Yaskawa INFORM job: A_ROOF_SIDE_0617_2_PAINT_44.JBI

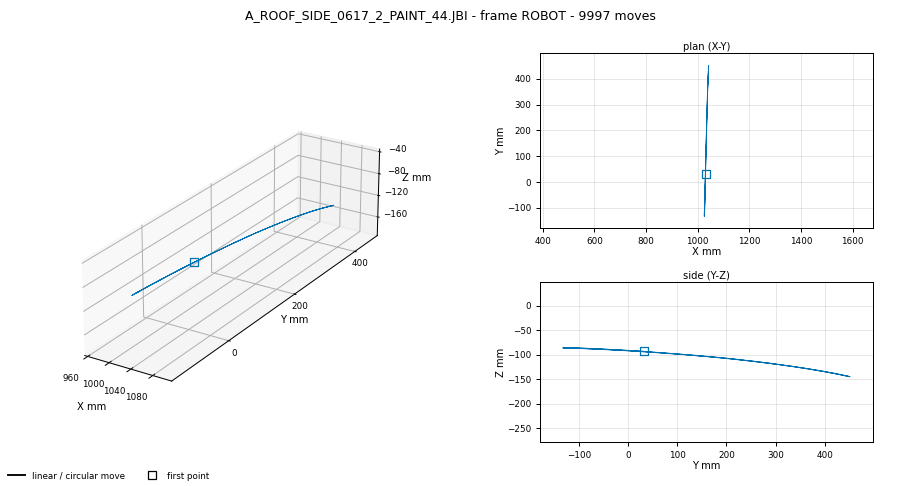
[picture p0: tool path of A_ROOF_SIDE_0617_2_PAINT_44.JBI in frame ROBOT, 9997 of 9997 moves have a stored position in this frame; points joined in program order, loops and branches not executed]
/JOB
//NAME A_ROOF_SIDE_0617_2_PAINT44
//POS
///NPOS 9997,0,0,0,0,0
///TOOL 1
///USER 0
///POSTYPE ROBOT
///RECTAN
///RCONF 1,0,0,0,0,0,0,0,0,0,0,0,0,0,0,0,0,0,0,0,0,0,0,0
C00000=1030.826,31.306,-92.980,168.331,43.416,158.095
C00001=1030.820,31.056,-92.964,168.328,43.418,158.095
C00002=1030.814,30.807,-92.948,168.325,43.419,158.095
C00003=1030.807,30.558,-92.932,168.324,43.421,158.095
C00004=1030.801,30.309,-92.916,168.321,43.422,158.095
C00005=1030.795,30.059,-92.899,168.319,43.423,158.096
C00006=1030.788,29.809,-92.884,168.316,43.425,158.096
C00007=1030.782,29.560,-92.868,168.314,43.426,158.096
C00008=1030.776,29.310,-92.852,168.312,43.427,158.096
C00009=1030.770,29.061,-92.836,168.309,43.429,158.096
C00010=1030.764,28.812,-92.820,168.306,43.431,158.096
C00011=1030.758,28.562,-92.803,168.305,43.432,158.096
C00012=1030.750,28.276,-92.785,168.302,43.433,158.096
C00013=1030.744,27.990,-92.767,168.299,43.435,158.096
C00014=1030.737,27.704,-92.749,168.297,43.437,158.096
C00015=1030.728,27.418,-92.731,168.294,43.438,158.096
C00016=1030.722,27.169,-92.714,168.291,43.440,158.096
C00017=1030.716,26.919,-92.699,168.289,43.442,158.097
C00018=1030.710,26.670,-92.683,168.287,43.443,158.097
C00019=1030.703,26.421,-92.667,168.284,43.445,158.097
C00020=1030.697,26.171,-92.651,168.281,43.446,158.097
C00021=1030.692,25.921,-92.636,168.280,43.448,158.097
C00022=1030.685,25.672,-92.620,168.277,43.449,158.097
C00023=1030.678,25.422,-92.604,168.274,43.451,158.097
C00024=1030.672,25.173,-92.588,168.272,43.452,158.097
C00025=1030.665,24.923,-92.573,168.270,43.454,158.097
C00026=1030.660,24.674,-92.556,168.267,43.456,158.097
C00027=1030.653,24.425,-92.541,168.265,43.457,158.097
C00028=1030.647,24.175,-92.525,168.263,43.459,158.098
C00029=1030.641,23.926,-92.510,168.260,43.460,158.098
C00030=1030.635,23.677,-92.493,168.257,43.462,158.098
C00031=1030.628,23.427,-92.478,168.255,43.463,158.098
C00032=1030.622,23.178,-92.462,168.253,43.464,158.098
C00033=1030.616,22.929,-92.446,168.250,43.466,158.098
C00034=1030.610,22.679,-92.431,168.248,43.467,158.098
C00035=1030.603,22.430,-92.415,168.245,43.469,158.098
C00036=1030.597,22.181,-92.400,168.243,43.470,158.098
C00037=1030.591,21.931,-92.384,168.241,43.471,158.098
C00038=1030.584,21.682,-92.368,168.238,43.473,158.098
C00039=1030.579,21.432,-92.353,168.236,43.474,158.098
C00040=1030.572,21.183,-92.337,168.234,43.476,158.098
C00041=1030.566,20.933,-92.321,168.231,43.477,158.098
C00042=1030.560,20.684,-92.306,168.228,43.479,158.099
C00043=1030.554,20.434,-92.290,168.227,43.480,158.099
C00044=1030.547,20.185,-92.275,168.224,43.482,158.099
C00045=1030.540,19.936,-92.259,168.221,43.483,158.099
C00046=1030.535,19.686,-92.244,168.220,43.485,158.099
C00047=1030.528,19.437,-92.228,168.217,43.487,158.099
C00048=1030.523,19.187,-92.212,168.214,43.488,158.099
C00049=1030.516,18.938,-92.197,168.212,43.490,158.099
C00050=1030.509,18.688,-92.182,168.210,43.491,158.099
C00051=1030.503,18.439,-92.166,168.207,43.493,158.099
C00052=1030.497,18.189,-92.151,168.204,43.494,158.099
C00053=1030.490,17.940,-92.135,168.203,43.496,158.100
C00054=1030.484,17.690,-92.120,168.200,43.498,158.100
C00055=1030.478,17.441,-92.104,168.197,43.499,158.100
C00056=1030.472,17.191,-92.089,168.195,43.500,158.100
C00057=1030.465,16.942,-92.074,168.193,43.502,158.100
C00058=1030.459,16.692,-92.058,168.190,43.504,158.100
C00059=1030.453,16.442,-92.043,168.188,43.505,158.100
C00060=1030.446,16.193,-92.027,168.186,43.506,158.100
C00061=1030.440,15.944,-92.012,168.183,43.508,158.100
C00062=1030.434,15.694,-91.996,168.180,43.509,158.100
C00063=1030.428,15.445,-91.981,168.178,43.511,158.100
C00064=1030.421,15.195,-91.966,168.176,43.512,158.100
C00065=1030.416,14.947,-91.950,168.173,43.514,158.101
C00066=1030.409,14.697,-91.935,168.171,43.515,158.101
C00067=1030.403,14.447,-91.920,168.169,43.517,158.101
C00068=1030.396,14.198,-91.904,168.166,43.518,158.101
C00069=1030.391,13.948,-91.889,168.164,43.520,158.101
C00070=1030.384,13.699,-91.874,168.161,43.521,158.101
C00071=1030.378,13.449,-91.858,168.159,43.523,158.101
C00072=1030.371,13.200,-91.843,168.156,43.525,158.101
C00073=1030.365,12.950,-91.828,168.154,43.526,158.101
C00074=1030.359,12.701,-91.813,168.151,43.528,158.101
C00075=1030.352,12.451,-91.798,168.149,43.530,158.101
C00076=1030.345,12.166,-91.781,168.146,43.531,158.101
C00077=1030.338,11.882,-91.764,168.143,43.533,158.102
C00078=1030.330,11.597,-91.747,168.141,43.535,158.102
C00079=1030.323,11.312,-91.729,168.137,43.537,158.102
C00080=1030.317,11.063,-91.715,168.136,43.538,158.102
C00081=1030.310,10.813,-91.700,168.133,43.540,158.102
C00082=1030.304,10.563,-91.685,168.130,43.541,158.102
C00083=1030.298,10.314,-91.670,168.127,43.543,158.102
C00084=1030.291,10.065,-91.654,168.126,43.544,158.102
C00085=1030.285,9.816,-91.639,168.123,43.546,158.102
C00086=1030.279,9.566,-91.624,168.120,43.548,158.103
C00087=1030.272,9.317,-91.610,168.117,43.549,158.102
C00088=1030.266,9.067,-91.595,168.116,43.551,158.103
C00089=1030.260,8.817,-91.580,168.113,43.553,158.103
C00090=1030.253,8.568,-91.565,168.110,43.554,158.103
C00091=1030.247,8.319,-91.550,168.108,43.556,158.103
C00092=1030.241,8.069,-91.535,168.105,43.558,158.103
C00093=1030.234,7.820,-91.520,168.103,43.559,158.103
C00094=1030.228,7.570,-91.505,168.101,43.561,158.103
C00095=1030.222,7.321,-91.490,168.098,43.562,158.103
C00096=1030.215,7.071,-91.475,168.095,43.564,158.103
C00097=1030.209,6.822,-91.460,168.094,43.566,158.104
C00098=1030.203,6.572,-91.445,168.091,43.567,158.104
C00099=1030.197,6.323,-91.430,168.088,43.569,158.104
C00100=1030.190,6.073,-91.415,168.085,43.570,158.104
C00101=1030.184,5.824,-91.401,168.084,43.572,158.104
C00102=1030.178,5.574,-91.386,168.081,43.573,158.104
C00103=1030.172,5.325,-91.371,168.078,43.575,158.104
C00104=1030.165,5.075,-91.356,168.076,43.576,158.104
C00105=1030.159,4.825,-91.341,168.074,43.577,158.104
C00106=1030.153,4.576,-91.326,168.071,43.579,158.104
C00107=1030.147,4.327,-91.311,168.068,43.581,158.104
C00108=1030.140,4.077,-91.296,168.066,43.582,158.104
C00109=1030.134,3.827,-91.281,168.063,43.584,158.104
C00110=1030.128,3.579,-91.267,168.061,43.585,158.104
C00111=1030.122,3.329,-91.252,168.059,43.587,158.105
C00112=1030.115,3.079,-91.237,168.056,43.588,158.105
C00113=1030.110,2.830,-91.222,168.053,43.590,158.105
C00114=1030.103,2.581,-91.207,168.051,43.592,158.105
C00115=1030.097,2.331,-91.193,168.049,43.593,158.105
C00116=1030.090,2.081,-91.178,168.046,43.595,158.105
C00117=1030.085,1.832,-91.164,168.043,43.596,158.105
C00118=1030.079,1.582,-91.149,168.042,43.598,158.105
C00119=1030.072,1.332,-91.134,168.039,43.599,158.105
C00120=1030.066,1.083,-91.119,168.036,43.601,158.105
C00121=1030.060,0.834,-91.104,168.033,43.602,158.105
C00122=1030.054,0.584,-91.089,168.032,43.604,158.105
C00123=1030.048,0.335,-91.075,168.029,43.605,158.105
C00124=1030.042,0.086,-91.060,168.026,43.607,158.106
C00125=1030.035,-0.165,-91.046,168.023,43.608,158.106
C00126=1030.030,-0.414,-91.031,168.021,43.610,158.106
C00127=1030.023,-0.663,-91.017,168.019,43.612,158.106
C00128=1030.016,-0.913,-91.002,168.016,43.613,158.106
C00129=1030.010,-1.162,-90.987,168.014,43.615,158.106
C00130=1030.004,-1.411,-90.972,168.011,43.616,158.106
C00131=1029.999,-1.661,-90.958,168.009,43.618,158.106
C00132=1029.992,-1.911,-90.943,168.006,43.619,158.106
C00133=1029.986,-2.160,-90.928,168.004,43.621,158.106
C00134=1029.980,-2.409,-90.914,168.001,43.622,158.106
C00135=1029.974,-2.659,-90.899,167.999,43.624,158.106
C00136=1029.968,-2.908,-90.885,167.996,43.625,158.106
C00137=1029.962,-3.158,-90.870,167.994,43.627,158.107
C00138=1029.955,-3.408,-90.855,167.991,43.628,158.107
C00139=1029.950,-3.657,-90.841,167.989,43.630,158.107
C00140=1029.942,-3.940,-90.824,167.985,43.631,158.107
C00141=1029.935,-4.223,-90.809,167.983,43.633,158.107
C00142=1029.928,-4.505,-90.792,167.980,43.635,158.107
C00143=1029.921,-4.789,-90.775,167.978,43.637,158.107
C00144=1029.915,-5.038,-90.762,167.975,43.639,158.107
C00145=1029.908,-5.288,-90.747,167.972,43.641,158.107
C00146=1029.902,-5.537,-90.733,167.969,43.642,158.107
C00147=1029.896,-5.787,-90.719,167.967,43.644,158.107
C00148=1029.889,-6.036,-90.704,167.964,43.646,158.107
C00149=1029.883,-6.286,-90.691,167.962,43.647,158.108
C00150=1029.877,-6.535,-90.676,167.960,43.649,158.108
C00151=1029.871,-6.784,-90.661,167.957,43.650,158.108
C00152=1029.864,-7.034,-90.648,167.954,43.652,158.108
C00153=1029.858,-7.284,-90.633,167.952,43.654,158.108
C00154=1029.851,-7.533,-90.619,167.949,43.655,158.108
C00155=1029.845,-7.783,-90.604,167.946,43.657,158.108
C00156=1029.840,-8.032,-90.591,167.945,43.658,158.108
C00157=1029.832,-8.282,-90.576,167.942,43.660,158.108
C00158=1029.827,-8.531,-90.562,167.939,43.661,158.108
C00159=1029.820,-8.781,-90.548,167.936,43.663,158.108
C00160=1029.814,-9.030,-90.534,167.934,43.665,158.109
C00161=1029.808,-9.280,-90.519,167.931,43.666,158.109
C00162=1029.801,-9.530,-90.506,167.928,43.668,158.109
C00163=1029.795,-9.779,-90.491,167.927,43.670,158.109
C00164=1029.789,-10.029,-90.477,167.924,43.671,158.109
C00165=1029.783,-10.278,-90.463,167.921,43.673,158.109
C00166=1029.776,-10.528,-90.449,167.919,43.675,158.109
C00167=1029.770,-10.777,-90.435,167.916,43.676,158.109
C00168=1029.764,-11.027,-90.420,167.913,43.678,158.109
C00169=1029.758,-11.276,-90.407,167.911,43.680,158.109
C00170=1029.752,-11.526,-90.392,167.909,43.681,158.109
C00171=1029.745,-11.775,-90.379,167.906,43.683,158.109
C00172=1029.740,-12.025,-90.365,167.903,43.684,158.109
C00173=1029.733,-12.274,-90.351,167.901,43.686,158.110
C00174=1029.727,-12.524,-90.337,167.898,43.688,158.110
C00175=1029.721,-12.773,-90.322,167.895,43.689,158.110
C00176=1029.715,-13.023,-90.309,167.893,43.691,158.110
C00177=1029.709,-13.273,-90.294,167.891,43.693,158.110
C00178=1029.702,-13.521,-90.280,167.888,43.694,158.110
C00179=1029.696,-13.772,-90.266,167.885,43.696,158.110
C00180=1029.690,-14.021,-90.253,167.883,43.697,158.110
C00181=1029.684,-14.270,-90.238,167.880,43.699,158.110
C00182=1029.678,-14.520,-90.224,167.877,43.701,158.110
C00183=1029.672,-14.770,-90.211,167.875,43.702,158.110
C00184=1029.666,-15.020,-90.197,167.873,43.704,158.110
C00185=1029.659,-15.268,-90.183,167.870,43.705,158.110
C00186=1029.653,-15.519,-90.168,167.867,43.707,158.111
C00187=1029.647,-15.768,-90.155,167.865,43.709,158.111
C00188=1029.640,-16.018,-90.141,167.862,43.710,158.111
C00189=1029.634,-16.267,-90.127,167.859,43.712,158.111
C00190=1029.628,-16.516,-90.114,167.857,43.714,158.111
C00191=1029.621,-16.766,-90.100,167.854,43.716,158.111
C00192=1029.616,-17.016,-90.086,167.851,43.717,158.111
C00193=1029.609,-17.266,-90.072,167.849,43.719,158.111
C00194=1029.603,-17.515,-90.059,167.847,43.720,158.111
C00195=1029.597,-17.764,-90.045,167.844,43.722,158.111
C00196=1029.590,-18.014,-90.031,167.842,43.723,158.111
C00197=1029.584,-18.263,-90.018,167.839,43.725,158.112
C00198=1029.578,-18.513,-90.003,167.836,43.727,158.112
C00199=1029.572,-18.763,-89.990,167.834,43.729,158.112
C00200=1029.565,-19.012,-89.977,167.831,43.730,158.112
C00201=1029.559,-19.262,-89.963,167.828,43.732,158.112
C00202=1029.553,-19.511,-89.949,167.826,43.734,158.112
C00203=1029.547,-19.761,-89.936,167.823,43.736,158.112
C00204=1029.540,-20.042,-89.920,167.820,43.738,158.112
C00205=1029.533,-20.323,-89.905,167.817,43.739,158.112
C00206=1029.525,-20.605,-89.890,167.814,43.741,158.112
C00207=1029.518,-20.886,-89.874,167.811,43.743,158.112
C00208=1029.512,-21.135,-89.861,167.809,43.745,158.113
C00209=1029.506,-21.385,-89.847,167.806,43.747,158.113
C00210=1029.500,-21.635,-89.833,167.803,43.748,158.113
C00211=1029.493,-21.884,-89.820,167.800,43.750,158.113
C00212=1029.487,-22.134,-89.807,167.798,43.752,158.113
C00213=1029.482,-22.383,-89.793,167.795,43.754,158.113
C00214=1029.475,-22.633,-89.779,167.793,43.755,158.113
C00215=1029.469,-22.882,-89.766,167.791,43.757,158.113
C00216=1029.463,-23.132,-89.752,167.788,43.759,158.113
C00217=1029.456,-23.382,-89.739,167.785,43.760,158.113
C00218=1029.450,-23.631,-89.725,167.783,43.762,158.113
C00219=1029.444,-23.880,-89.712,167.780,43.764,158.113
C00220=1029.438,-24.130,-89.698,167.777,43.765,158.113
C00221=1029.432,-24.380,-89.684,167.775,43.767,158.114
C00222=1029.425,-24.629,-89.671,167.772,43.769,158.114
C00223=1029.419,-24.878,-89.658,167.769,43.770,158.114
C00224=1029.414,-25.128,-89.644,167.766,43.772,158.114
C00225=1029.407,-25.378,-89.630,167.764,43.774,158.114
C00226=1029.401,-25.628,-89.618,167.761,43.775,158.114
C00227=1029.395,-25.877,-89.605,167.758,43.777,158.114
C00228=1029.389,-26.127,-89.591,167.756,43.779,158.114
C00229=1029.383,-26.376,-89.577,167.754,43.780,158.114
C00230=1029.376,-26.626,-89.564,167.751,43.782,158.114
C00231=1029.370,-26.875,-89.551,167.749,43.783,158.114
C00232=1029.365,-27.125,-89.537,167.746,43.785,158.114
C00233=1029.359,-27.375,-89.524,167.743,43.787,158.115
C00234=1029.352,-27.625,-89.511,167.741,43.788,158.115
C00235=1029.346,-27.874,-89.497,167.738,43.790,158.115
C00236=1029.339,-28.123,-89.484,167.735,43.792,158.115
C00237=1029.334,-28.373,-89.471,167.732,43.793,158.115
C00238=1029.327,-28.622,-89.458,167.730,43.795,158.115
C00239=1029.321,-28.872,-89.445,167.727,43.797,158.115
C00240=1029.314,-29.122,-89.431,167.725,43.799,158.115
C00241=1029.308,-29.371,-89.419,167.722,43.801,158.115
C00242=1029.302,-29.621,-89.405,167.719,43.802,158.115
C00243=1029.296,-29.870,-89.392,167.716,43.804,158.115
C00244=1029.289,-30.121,-89.379,167.714,43.806,158.116
C00245=1029.283,-30.370,-89.366,167.711,43.808,158.116
C00246=1029.277,-30.619,-89.353,167.709,43.810,158.116
C00247=1029.271,-30.869,-89.340,167.706,43.811,158.116
C00248=1029.265,-31.118,-89.327,167.703,43.813,158.116
C00249=1029.259,-31.367,-89.314,167.701,43.815,158.116
C00250=1029.253,-31.617,-89.301,167.698,43.817,158.116
C00251=1029.246,-31.867,-89.287,167.695,43.818,158.116
C00252=1029.240,-32.117,-89.274,167.692,43.820,158.116
C00253=1029.234,-32.366,-89.262,167.690,43.822,158.116
C00254=1029.228,-32.616,-89.248,167.687,43.824,158.116
C00255=1029.222,-32.866,-89.236,167.685,43.826,158.117
C00256=1029.216,-33.115,-89.223,167.682,43.827,158.117
C00257=1029.209,-33.364,-89.209,167.679,43.829,158.117
C00258=1029.203,-33.614,-89.197,167.676,43.831,158.117
C00259=1029.196,-33.864,-89.184,167.674,43.833,158.117
C00260=1029.190,-34.114,-89.171,167.671,43.834,158.117
C00261=1029.184,-34.363,-89.158,167.668,43.836,158.117
C00262=1029.178,-34.613,-89.145,167.666,43.838,158.117
C00263=1029.172,-34.862,-89.132,167.663,43.840,158.117
C00264=1029.166,-35.112,-89.119,167.660,43.841,158.117
C00265=1029.159,-35.361,-89.106,167.658,43.843,158.117
C00266=1029.154,-35.611,-89.094,167.655,43.845,158.117
C00267=1029.147,-35.860,-89.080,167.652,43.846,158.118
C00268=1029.141,-36.141,-89.066,167.649,43.849,158.118
C00269=1029.134,-36.421,-89.052,167.646,43.850,158.118
C00270=1029.127,-36.702,-89.037,167.643,43.852,158.118
C00271=1029.120,-36.982,-89.023,167.640,43.854,158.118
C00272=1029.114,-37.232,-89.010,167.637,43.856,158.118
C00273=1029.108,-37.481,-88.997,167.634,43.858,158.118
C00274=1029.102,-37.731,-88.984,167.632,43.859,158.118
C00275=1029.095,-37.980,-88.971,167.629,43.861,158.118
C00276=1029.090,-38.230,-88.958,167.626,43.863,158.118
C00277=1029.084,-38.480,-88.946,167.624,43.864,158.118
C00278=1029.077,-38.729,-88.933,167.621,43.866,158.118
C00279=1029.072,-38.979,-88.920,167.618,43.868,158.118
C00280=1029.065,-39.228,-88.907,167.616,43.870,158.119
C00281=1029.059,-39.478,-88.895,167.613,43.871,158.119
C00282=1029.053,-39.728,-88.882,167.610,43.873,158.119
C00283=1029.047,-39.978,-88.870,167.608,43.875,158.119
C00284=1029.040,-40.227,-88.857,167.605,43.877,158.119
C00285=1029.034,-40.476,-88.845,167.602,43.879,158.119
C00286=1029.028,-40.726,-88.832,167.600,43.881,158.119
C00287=1029.022,-40.976,-88.819,167.596,43.882,158.119
C00288=1029.015,-41.225,-88.807,167.593,43.884,158.119
C00289=1029.009,-41.475,-88.794,167.591,43.886,158.119
C00290=1029.003,-41.725,-88.782,167.588,43.888,158.119
C00291=1028.996,-41.974,-88.769,167.585,43.890,158.120
C00292=1028.991,-42.224,-88.756,167.583,43.892,158.120
C00293=1028.985,-42.474,-88.744,167.580,43.894,158.120
C00294=1028.978,-42.723,-88.732,167.578,43.896,158.120
C00295=1028.972,-42.973,-88.719,167.575,43.897,158.120
C00296=1028.966,-43.222,-88.706,167.572,43.899,158.120
C00297=1028.959,-43.472,-88.694,167.569,43.901,158.120
C00298=1028.953,-43.722,-88.682,167.567,43.903,158.120
C00299=1028.948,-43.971,-88.669,167.563,43.905,158.120
C00300=1028.941,-44.221,-88.657,167.561,43.907,158.120
C00301=1028.935,-44.471,-88.645,167.558,43.909,158.121
C00302=1028.929,-44.720,-88.632,167.555,43.910,158.120
C00303=1028.923,-44.969,-88.620,167.552,43.912,158.121
C00304=1028.917,-45.219,-88.607,167.550,43.914,158.121
C00305=1028.911,-45.469,-88.595,167.547,43.916,158.121
C00306=1028.904,-45.719,-88.583,167.545,43.917,158.121
C00307=1028.898,-45.969,-88.570,167.542,43.919,158.121
C00308=1028.893,-46.218,-88.558,167.539,43.921,158.121
C00309=1028.886,-46.467,-88.546,167.536,43.923,158.121
C00310=1028.880,-46.717,-88.533,167.534,43.924,158.121
C00311=1028.874,-46.966,-88.520,167.531,43.926,158.121
C00312=1028.867,-47.216,-88.508,167.528,43.928,158.121
C00313=1028.862,-47.466,-88.496,167.525,43.930,158.122
C00314=1028.856,-47.715,-88.483,167.522,43.932,158.122
C00315=1028.850,-47.965,-88.471,167.520,43.933,158.122
C00316=1028.844,-48.215,-88.459,167.517,43.935,158.122
C00317=1028.838,-48.464,-88.446,167.514,43.937,158.122
C00318=1028.831,-48.714,-88.434,167.512,43.939,158.122
C00319=1028.826,-48.963,-88.422,167.509,43.940,158.122
C00320=1028.819,-49.213,-88.410,167.506,43.942,158.122
C00321=1028.813,-49.463,-88.398,167.504,43.944,158.122
C00322=1028.807,-49.713,-88.385,167.501,43.946,158.122
C00323=1028.801,-49.962,-88.373,167.498,43.948,158.122
C00324=1028.795,-50.211,-88.361,167.494,43.950,158.122
C00325=1028.790,-50.461,-88.348,167.492,43.951,158.122
C00326=1028.783,-50.711,-88.336,167.489,43.953,158.123
C00327=1028.777,-50.961,-88.325,167.487,43.955,158.123
C00328=1028.771,-51.211,-88.313,167.484,43.957,158.123
C00329=1028.765,-51.460,-88.301,167.481,43.959,158.123
C00330=1028.758,-51.709,-88.289,167.479,43.961,158.123
C00331=1028.752,-51.959,-88.276,167.475,43.963,158.123
C00332=1028.743,-52.314,-88.260,167.472,43.966,158.123
C00333=1028.734,-52.667,-88.243,167.467,43.969,158.123
C00334=1028.725,-53.021,-88.226,167.464,43.972,158.124
C00335=1028.717,-53.376,-88.209,167.459,43.975,158.124
C00336=1028.710,-53.625,-88.197,167.457,43.977,158.124
C00337=1028.704,-53.874,-88.186,167.454,43.978,158.124
C00338=1028.698,-54.124,-88.175,167.451,43.980,158.124
C00339=1028.692,-54.374,-88.162,167.449,43.982,158.124
C00340=1028.685,-54.624,-88.150,167.445,43.984,158.124
C00341=1028.679,-54.873,-88.139,167.443,43.986,158.124
C00342=1028.673,-55.123,-88.127,167.440,43.988,158.124
C00343=1028.667,-55.373,-88.115,167.437,43.990,158.125
C00344=1028.661,-55.622,-88.103,167.435,43.992,158.125
C00345=1028.654,-55.872,-88.092,167.431,43.994,158.125
C00346=1028.648,-56.121,-88.080,167.428,43.996,158.125
C00347=1028.642,-56.371,-88.068,167.426,43.998,158.125
C00348=1028.636,-56.621,-88.057,167.423,44.000,158.125
C00349=1028.629,-56.870,-88.045,167.421,44.002,158.125
C00350=1028.623,-57.120,-88.033,167.417,44.004,158.125
C00351=1028.618,-57.370,-88.021,167.414,44.006,158.125
C00352=1028.611,-57.619,-88.009,167.412,44.008,158.125
C00353=1028.605,-57.869,-87.998,167.409,44.010,158.126
C00354=1028.599,-58.118,-87.986,167.406,44.012,158.126
C00355=1028.593,-58.369,-87.974,167.404,44.014,158.126
C00356=1028.587,-58.618,-87.963,167.400,44.016,158.126
C00357=1028.580,-58.867,-87.951,167.397,44.018,158.126
C00358=1028.574,-59.117,-87.940,167.395,44.019,158.126
C00359=1028.568,-59.366,-87.928,167.392,44.021,158.126
C00360=1028.562,-59.617,-87.916,167.390,44.023,158.126
C00361=1028.556,-59.866,-87.904,167.386,44.025,158.126
C00362=1028.550,-60.116,-87.893,167.383,44.027,158.126
C00363=1028.543,-60.365,-87.881,167.381,44.029,158.126
C00364=1028.538,-60.615,-87.870,167.378,44.031,158.127
C00365=1028.532,-60.865,-87.858,167.375,44.033,158.127
C00366=1028.526,-61.114,-87.847,167.372,44.035,158.127
C00367=1028.519,-61.364,-87.835,167.369,44.037,158.127
C00368=1028.513,-61.614,-87.824,167.367,44.039,158.127
C00369=1028.508,-61.863,-87.812,167.364,44.041,158.127
C00370=1028.501,-62.113,-87.801,167.361,44.043,158.127
C00371=1028.495,-62.362,-87.789,167.358,44.045,158.127
C00372=1028.489,-62.613,-87.778,167.355,44.047,158.127
C00373=1028.483,-62.861,-87.766,167.352,44.049,158.127
C00374=1028.477,-63.112,-87.754,167.350,44.051,158.128
C00375=1028.471,-63.361,-87.743,167.347,44.053,158.128
C00376=1028.465,-63.611,-87.731,167.344,44.055,158.128
C00377=1028.459,-63.860,-87.721,167.341,44.057,158.128
C00378=1028.453,-64.110,-87.709,167.338,44.059,158.128
C00379=1028.448,-64.360,-87.697,167.336,44.061,158.128
C00380=1028.441,-64.609,-87.685,167.333,44.063,158.128
C00381=1028.435,-64.859,-87.674,167.330,44.064,158.128
C00382=1028.429,-65.109,-87.663,167.327,44.067,158.128
C00383=1028.423,-65.358,-87.651,167.324,44.068,158.128
C00384=1028.417,-65.608,-87.640,167.322,44.070,158.129
C00385=1028.412,-65.858,-87.629,167.319,44.072,158.129
C00386=1028.405,-66.107,-87.617,167.316,44.074,158.129
C00387=1028.399,-66.357,-87.606,167.313,44.076,158.129
C00388=1028.393,-66.570,-87.596,167.311,44.077,158.129
C00389=1028.389,-66.783,-87.586,167.308,44.079,158.129
C00390=1028.384,-66.997,-87.577,167.306,44.081,158.129
C00391=1028.379,-67.209,-87.567,167.303,44.083,158.129
C00392=1028.373,-67.423,-87.557,167.301,44.084,158.129
C00393=1028.368,-67.636,-87.547,167.299,44.086,158.129
C00394=1028.364,-67.849,-87.538,167.296,44.087,158.129
C00395=1028.358,-68.062,-87.528,167.294,44.089,158.129
C00396=1028.352,-68.344,-87.516,167.290,44.091,158.129
C00397=1028.345,-68.626,-87.502,167.287,44.093,158.130
C00398=1028.338,-68.908,-87.490,167.284,44.096,158.130
C00399=1028.331,-69.191,-87.477,167.281,44.098,158.130
C00400=1028.325,-69.440,-87.466,167.278,44.100,158.130
C00401=1028.320,-69.690,-87.455,167.275,44.102,158.130
///RCONF 1,0,0,1,0,0,0,0,0,0,0,0,0,0,0,0,0,0,0,0,0,0,0,0
C00402=1028.314,-69.940,-87.443,167.272,44.104,158.130
C00403=1028.308,-70.189,-87.432,167.269,44.106,158.130
C00404=1028.302,-70.439,-87.421,167.266,44.107,158.130
C00405=1028.296,-70.689,-87.410,167.264,44.109,158.130
C00406=1028.290,-70.938,-87.399,167.261,44.111,158.130
C00407=1028.284,-71.188,-87.388,167.257,44.113,158.130
C00408=1028.278,-71.437,-87.376,167.255,44.115,158.130
C00409=1028.273,-71.687,-87.365,167.252,44.117,158.131
C00410=1028.267,-71.937,-87.354,167.250,44.119,158.131
C00411=1028.261,-72.187,-87.342,167.247,44.121,158.131
C00412=1028.255,-72.436,-87.332,167.243,44.123,158.131
C00413=1028.249,-72.686,-87.321,167.241,44.125,158.131
C00414=1028.243,-72.936,-87.309,167.238,44.127,158.131
C00415=1028.237,-73.185,-87.299,167.235,44.129,158.131
C00416=1028.232,-73.435,-87.287,167.233,44.131,158.131
C00417=1028.225,-73.685,-87.275,167.229,44.132,158.131
C00418=1028.220,-73.934,-87.264,167.226,44.134,158.131
C00419=1028.214,-74.184,-87.253,167.224,44.136,158.131
C00420=1028.208,-74.433,-87.243,167.221,44.138,158.131
C00421=1028.202,-74.684,-87.231,167.219,44.140,158.132
C00422=1028.196,-74.933,-87.220,167.215,44.143,158.132
C00423=1028.190,-75.182,-87.210,167.212,44.145,158.132
C00424=1028.184,-75.433,-87.200,167.210,44.147,158.132
C00425=1028.178,-75.682,-87.189,167.206,44.149,158.132
C00426=1028.172,-75.932,-87.178,167.204,44.151,158.132
C00427=1028.166,-76.181,-87.167,167.201,44.153,158.132
C00428=1028.160,-76.432,-87.156,167.198,44.155,158.132
C00429=1028.154,-76.681,-87.145,167.195,44.157,158.132
C00430=1028.148,-76.930,-87.135,167.192,44.159,158.132
C00431=1028.141,-77.181,-87.123,167.189,44.161,158.133
C00432=1028.136,-77.430,-87.112,167.187,44.163,158.133
C00433=1028.130,-77.679,-87.102,167.183,44.165,158.133
C00434=1028.125,-77.930,-87.091,167.181,44.167,158.133
C00435=1028.119,-78.179,-87.080,167.178,44.169,158.133
C00436=1028.112,-78.429,-87.070,167.175,44.171,158.133
C00437=1028.106,-78.678,-87.059,167.172,44.173,158.133
C00438=1028.100,-78.928,-87.048,167.169,44.175,158.133
C00439=1028.094,-79.177,-87.037,167.167,44.177,158.133
C00440=1028.088,-79.428,-87.027,167.163,44.179,158.133
C00441=1028.083,-79.678,-87.016,167.160,44.181,158.134
C00442=1028.076,-79.927,-87.006,167.158,44.183,158.134
C00443=1028.070,-80.176,-86.995,167.154,44.186,158.134
C00444=1028.065,-80.427,-86.984,167.152,44.188,158.134
C00445=1028.058,-80.676,-86.974,167.149,44.190,158.134
C00446=1028.052,-80.926,-86.963,167.145,44.192,158.134
C00447=1028.046,-81.176,-86.953,167.143,44.195,158.134
C00448=1028.040,-81.425,-86.943,167.140,44.196,158.134
C00449=1028.035,-81.675,-86.932,167.137,44.199,158.135
C00450=1028.028,-81.925,-86.922,167.134,44.201,158.135
C00451=1028.022,-82.175,-86.911,167.132,44.203,158.135
C00452=1028.016,-82.424,-86.901,167.128,44.205,158.135
C00453=1028.010,-82.674,-86.890,167.126,44.207,158.135
C00454=1028.004,-82.923,-86.880,167.123,44.210,158.135
C00455=1027.998,-83.173,-86.870,167.119,44.212,158.135
C00456=1027.992,-83.423,-86.859,167.117,44.214,158.135
C00457=1027.985,-83.673,-86.848,167.114,44.216,158.135
C00458=1027.980,-83.923,-86.838,167.111,44.219,158.136
C00459=1027.974,-84.172,-86.828,167.108,44.221,158.136
C00460=1027.967,-84.457,-86.816,167.105,44.223,158.136
C00461=1027.961,-84.740,-86.804,167.101,44.226,158.136
C00462=1027.953,-85.025,-86.793,167.099,44.228,158.136
C00463=1027.946,-85.309,-86.781,167.095,44.230,158.136
C00464=1027.941,-85.559,-86.770,167.091,44.232,158.136
C00465=1027.935,-85.809,-86.761,167.089,44.234,158.136
C00466=1027.929,-86.058,-86.750,167.086,44.237,158.137
C00467=1027.923,-86.308,-86.740,167.083,44.239,158.137
C00468=1027.917,-86.557,-86.729,167.080,44.241,158.137
C00469=1027.911,-86.807,-86.720,167.078,44.243,158.137
C00470=1027.905,-87.057,-86.709,167.074,44.246,158.137
C00471=1027.900,-87.307,-86.699,167.071,44.248,158.137
C00472=1027.893,-87.556,-86.689,167.069,44.250,158.137
C00473=1027.888,-87.806,-86.678,167.065,44.252,158.137
C00474=1027.881,-88.055,-86.668,167.063,44.255,158.138
C00475=1027.876,-88.305,-86.658,167.060,44.256,158.138
C00476=1027.870,-88.555,-86.648,167.057,44.259,158.138
C00477=1027.864,-88.805,-86.637,167.054,44.261,158.138
C00478=1027.858,-89.055,-86.628,167.052,44.263,158.138
C00479=1027.852,-89.304,-86.617,167.048,44.265,158.138
C00480=1027.846,-89.554,-86.607,167.045,44.267,158.138
C00481=1027.840,-89.804,-86.597,167.043,44.269,158.138
C00482=1027.834,-90.053,-86.587,167.039,44.271,158.138
C00483=1027.828,-90.303,-86.577,167.037,44.274,158.139
C00484=1027.822,-90.553,-86.567,167.034,44.276,158.139
C00485=1027.817,-90.803,-86.556,167.030,44.278,158.139
C00486=1027.810,-91.052,-86.547,167.028,44.280,158.139
C00487=1027.805,-91.302,-86.537,167.025,44.283,158.139
C00488=1027.798,-91.552,-86.526,167.022,44.285,158.139
C00489=1027.793,-91.802,-86.516,167.019,44.287,158.139
C00490=1027.787,-92.052,-86.507,167.016,44.289,158.139
C00491=1027.781,-92.301,-86.496,167.013,44.291,158.139
C00492=1027.775,-92.551,-86.486,167.010,44.293,158.140
C00493=1027.769,-92.801,-86.476,167.008,44.295,158.140
C00494=1027.763,-93.050,-86.466,167.004,44.298,158.140
C00495=1027.758,-93.300,-86.456,167.002,44.299,158.140
C00496=1027.751,-93.550,-86.446,166.999,44.301,158.140
C00497=1027.747,-93.799,-86.436,166.996,44.304,158.140
C00498=1027.740,-94.049,-86.426,166.993,44.306,158.140
C00499=1027.735,-94.299,-86.416,166.989,44.308,158.140
C00500=1027.728,-94.548,-86.406,166.987,44.310,158.140
C00501=1027.723,-94.799,-86.396,166.984,44.313,158.140
C00502=1027.717,-95.048,-86.387,166.981,44.315,158.141
C00503=1027.711,-95.298,-86.376,166.978,44.317,158.141
C00504=1027.705,-95.548,-86.366,166.975,44.319,158.141
C00505=1027.700,-95.797,-86.356,166.972,44.321,158.141
C00506=1027.694,-96.047,-86.347,166.969,44.324,158.141
C00507=1027.689,-96.297,-86.337,166.967,44.326,158.141
C00508=1027.682,-96.547,-86.327,166.963,44.328,158.141
C00509=1027.677,-96.796,-86.316,166.960,44.330,158.141
C00510=1027.671,-97.045,-86.307,166.958,44.332,158.141
C00511=1027.666,-97.295,-86.297,166.954,44.335,158.141
C00512=1027.659,-97.545,-86.287,166.952,44.337,158.142
C00513=1027.654,-97.795,-86.277,166.949,44.338,158.142
C00514=1027.648,-98.045,-86.267,166.946,44.341,158.142
C00515=1027.642,-98.295,-86.258,166.943,44.343,158.142
C00516=1027.636,-98.544,-86.249,166.939,44.345,158.142
C00517=1027.630,-98.794,-86.239,166.937,44.348,158.142
C00518=1027.624,-99.044,-86.229,166.934,44.350,158.142
C00519=1027.618,-99.294,-86.219,166.931,44.352,158.142
C00520=1027.612,-99.544,-86.210,166.928,44.355,158.143
C00521=1027.607,-99.793,-86.201,166.925,44.357,158.143
C00522=1027.601,-100.043,-86.190,166.922,44.360,158.143
C00523=1027.595,-100.293,-86.181,166.920,44.362,158.143
C00524=1027.588,-100.579,-86.170,166.916,44.364,158.143
C00525=1027.582,-100.866,-86.159,166.913,44.366,158.143
C00526=1027.575,-101.152,-86.148,166.909,44.369,158.143
C00527=1027.568,-101.439,-86.137,166.906,44.372,158.144
C00528=1027.563,-101.688,-86.128,166.903,44.374,158.144
C00529=1027.556,-101.938,-86.119,166.900,44.377,158.144
C00530=1027.550,-102.188,-86.109,166.897,44.379,158.144
C00531=1027.545,-102.438,-86.099,166.894,44.381,158.144
C00532=1027.539,-102.687,-86.090,166.891,44.384,158.144
C00533=1027.533,-102.937,-86.080,166.889,44.386,158.144
C00534=1027.527,-103.187,-86.071,166.885,44.388,158.144
C00535=1027.522,-103.436,-86.062,166.883,44.390,158.144
C00536=1027.515,-103.686,-86.053,166.879,44.393,158.145
C00537=1027.510,-103.936,-86.042,166.877,44.395,158.145
C00538=1027.504,-104.185,-86.033,166.874,44.397,158.145
C00539=1027.498,-104.435,-86.024,166.870,44.399,158.145
C00540=1027.492,-104.685,-86.015,166.868,44.402,158.145
C00541=1027.487,-104.935,-86.006,166.864,44.404,158.145
C00542=1027.481,-105.184,-85.996,166.862,44.407,158.145
C00543=1027.475,-105.434,-85.986,166.859,44.409,158.145
C00544=1027.470,-105.684,-85.977,166.856,44.411,158.146
C00545=1027.464,-105.934,-85.968,166.853,44.414,158.146
C00546=1027.458,-106.184,-85.958,166.850,44.416,158.146
///RCONF 1,0,0,0,0,0,0,0,0,0,0,0,0,0,0,0,0,0,0,0,0,0,0,0
C00547=1027.452,-106.433,-85.949,166.847,44.418,158.146
C00548=1027.446,-106.683,-85.940,166.844,44.421,158.146
C00549=1027.440,-106.933,-85.931,166.841,44.422,158.146
C00550=1027.434,-107.182,-85.921,166.838,44.425,158.146
C00551=1027.429,-107.433,-85.912,166.835,44.427,158.146
C00552=1027.423,-107.683,-85.902,166.832,44.430,158.147
C00553=1027.418,-107.932,-85.893,166.829,44.432,158.147
C00554=1027.412,-108.182,-85.884,166.826,44.435,158.147
C00555=1027.406,-108.431,-85.875,166.823,44.437,158.147
C00556=1027.400,-108.681,-85.866,166.820,44.440,158.147
C00557=1027.394,-108.932,-85.857,166.818,44.442,158.147
C00558=1027.389,-109.181,-85.848,166.814,44.444,158.147
C00559=1027.383,-109.431,-85.839,166.812,44.446,158.147
C00560=1027.377,-109.680,-85.829,166.808,44.449,158.148
C00561=1027.371,-109.930,-85.820,166.806,44.451,158.148
C00562=1027.365,-110.179,-85.812,166.802,44.454,158.148
C00563=1027.359,-110.429,-85.802,166.800,44.456,158.148
C00564=1027.353,-110.680,-85.794,166.796,44.459,158.148
C00565=1027.347,-110.929,-85.784,166.794,44.461,158.148
C00566=1027.341,-111.179,-85.776,166.791,44.463,158.149
C00567=1027.336,-111.428,-85.766,166.788,44.466,158.149
C00568=1027.330,-111.679,-85.757,166.785,44.468,158.149
C00569=1027.324,-111.928,-85.748,166.782,44.470,158.149
C00570=1027.319,-112.178,-85.739,166.779,44.473,158.149
C00571=1027.313,-112.427,-85.730,166.776,44.475,158.149
C00572=1027.307,-112.678,-85.721,166.773,44.478,158.149
C00573=1027.302,-112.927,-85.712,166.770,44.480,158.149
C00574=1027.296,-113.177,-85.703,166.767,44.482,158.149
C00575=1027.290,-113.426,-85.694,166.765,44.485,158.150
C00576=1027.284,-113.677,-85.685,166.761,44.487,158.150
C00577=1027.279,-113.926,-85.677,166.758,44.489,158.150
C00578=1027.273,-114.176,-85.667,166.755,44.492,158.150
C00579=1027.268,-114.426,-85.659,166.752,44.494,158.150
C00580=1027.261,-114.676,-85.649,166.749,44.496,158.150
C00581=1027.256,-114.925,-85.641,166.746,44.499,158.150
C00582=1027.250,-115.175,-85.632,166.743,44.502,158.151
C00583=1027.244,-115.425,-85.623,166.740,44.504,158.151
C00584=1027.238,-115.675,-85.614,166.738,44.507,158.151
C00585=1027.233,-115.925,-85.606,166.734,44.509,158.151
C00586=1027.227,-116.174,-85.597,166.732,44.511,158.151
C00587=1027.221,-116.424,-85.588,166.728,44.514,158.151
C00588=1027.215,-116.710,-85.578,166.725,44.516,158.151
C00589=1027.208,-116.996,-85.569,166.722,44.519,158.151
C00590=1027.202,-117.282,-85.558,166.718,44.522,158.152
C00591=1027.194,-117.568,-85.548,166.715,44.525,158.152
C00592=1027.189,-117.818,-85.539,166.712,44.528,158.152
C00593=1027.184,-118.068,-85.531,166.709,44.530,158.152
C00594=1027.177,-118.318,-85.523,166.706,44.533,158.152
C00595=1027.172,-118.567,-85.514,166.703,44.535,158.152
C00596=1027.166,-118.817,-85.505,166.700,44.537,158.153
C00597=1027.161,-119.067,-85.496,166.697,44.540,158.153
C00598=1027.155,-119.317,-85.488,166.694,44.542,158.153
C00599=1027.148,-119.566,-85.479,166.692,44.545,158.153
C00600=1027.143,-119.816,-85.470,166.688,44.548,158.153
C00601=1027.138,-120.066,-85.462,166.686,44.550,158.153
C00602=1027.132,-120.316,-85.453,166.682,44.553,158.153
C00603=1027.126,-120.565,-85.445,166.680,44.555,158.154
C00604=1027.121,-120.815,-85.437,166.676,44.557,158.154
C00605=1027.115,-121.066,-85.428,166.674,44.559,158.154
C00606=1027.109,-121.315,-85.418,166.670,44.562,158.154
C00607=1027.103,-121.564,-85.411,166.668,44.565,158.154
C00608=1027.097,-121.814,-85.402,166.664,44.567,158.154
C00609=1027.092,-122.064,-85.393,166.662,44.570,158.154
C00610=1027.086,-122.314,-85.385,166.659,44.573,158.155
C00611=1027.080,-122.564,-85.377,166.656,44.575,158.155
C00612=1027.075,-122.814,-85.368,166.653,44.577,158.155
C00613=1027.070,-123.063,-85.360,166.650,44.579,158.155
C00614=1027.064,-123.313,-85.352,166.646,44.582,158.155
C00615=1027.058,-123.563,-85.343,166.644,44.585,158.155
C00616=1027.053,-123.813,-85.334,166.640,44.587,158.155
C00617=1027.047,-124.062,-85.326,166.638,44.590,158.156
C00618=1027.041,-124.313,-85.318,166.635,44.592,158.156
C00619=1027.036,-124.563,-85.309,166.632,44.595,158.156
C00620=1027.030,-124.812,-85.301,166.630,44.597,158.156
C00621=1027.024,-125.062,-85.293,166.626,44.600,158.156
C00622=1027.018,-125.312,-85.284,166.624,44.602,158.156
C00623=1027.012,-125.561,-85.276,166.620,44.605,158.156
C00624=1027.007,-125.811,-85.267,166.618,44.608,158.157
C00625=1027.001,-126.061,-85.260,166.614,44.610,158.157
C00626=1026.995,-126.311,-85.251,166.612,44.613,158.157
C00627=1026.989,-126.560,-85.243,166.608,44.615,158.157
C00628=1026.984,-126.810,-85.234,166.606,44.617,158.157
C00629=1026.979,-127.060,-85.226,166.602,44.620,158.157
C00630=1026.973,-127.310,-85.219,166.600,44.623,158.158
C00631=1026.967,-127.560,-85.210,166.597,44.626,158.158
C00632=1026.961,-127.810,-85.202,166.594,44.628,158.158
C00633=1026.956,-128.058,-85.193,166.591,44.631,158.158
C00634=1026.951,-128.308,-85.185,166.588,44.633,158.158
C00635=1026.947,-128.558,-85.175,166.585,44.634,158.158
C00636=1026.943,-128.808,-85.165,166.582,44.634,158.158
C00637=1026.940,-129.057,-85.154,166.580,44.635,158.158
C00638=1026.938,-129.307,-85.142,166.577,44.635,158.157
C00639=1026.935,-129.557,-85.130,166.575,44.635,158.157
C00640=1026.934,-129.806,-85.119,166.573,44.634,158.157
C00641=1026.933,-130.057,-85.105,166.570,44.632,158.156
C00642=1026.933,-130.306,-85.092,166.569,44.630,158.156
C00643=1026.933,-130.556,-85.077,166.566,44.628,158.155
C00644=1026.934,-130.806,-85.062,166.564,44.625,158.154
C00645=1026.935,-131.056,-85.047,166.563,44.622,158.154
C00646=1026.938,-131.306,-85.031,166.560,44.618,158.153
C00647=1026.940,-131.555,-85.015,166.559,44.614,158.152
C00648=1026.943,-131.805,-84.997,166.557,44.609,158.151
C00649=1026.947,-132.056,-84.980,166.556,44.604,158.150
C00650=1026.951,-132.305,-84.962,166.555,44.598,158.149
C00651=1026.956,-132.555,-84.942,166.553,44.592,158.148
C00652=1026.648,-132.580,-85.262,166.504,44.850,158.186
C00653=1026.643,-132.331,-85.282,166.507,44.857,158.188
C00654=1026.639,-132.081,-85.300,166.507,44.863,158.189
C00655=1026.635,-131.831,-85.318,166.509,44.867,158.190
C00656=1026.632,-131.581,-85.334,166.511,44.872,158.191
C00657=1026.630,-131.331,-85.351,166.512,44.877,158.192
C00658=1026.628,-131.082,-85.368,166.515,44.881,158.193
C00659=1026.626,-130.831,-85.383,166.516,44.884,158.193
C00660=1026.626,-130.581,-85.398,166.518,44.887,158.194
C00661=1026.625,-130.332,-85.411,166.520,44.889,158.194
C00662=1026.625,-130.082,-85.425,166.522,44.891,158.195
C00663=1026.626,-129.832,-85.439,166.524,44.892,158.195
C00664=1026.628,-129.582,-85.451,166.527,44.893,158.196
C00665=1026.630,-129.333,-85.462,166.529,44.894,158.196
C00666=1026.632,-129.082,-85.474,166.532,44.894,158.196
C00667=1026.635,-128.833,-85.485,166.534,44.893,158.197
C00668=1026.639,-128.583,-85.495,166.537,44.892,158.197
C00669=1026.643,-128.334,-85.505,166.540,44.891,158.197
C00670=1026.648,-128.085,-85.514,166.542,44.889,158.197
C00671=1026.653,-127.835,-85.522,166.545,44.887,158.197
C00672=1026.659,-127.585,-85.530,166.548,44.884,158.196
C00673=1026.665,-127.336,-85.538,166.551,44.881,158.196
C00674=1026.670,-127.085,-85.547,166.554,44.878,158.196
C00675=1026.676,-126.836,-85.555,166.558,44.876,158.196
C00676=1026.682,-126.586,-85.564,166.560,44.873,158.196
C00677=1026.688,-126.337,-85.571,166.564,44.870,158.196
C00678=1026.693,-126.086,-85.579,166.566,44.868,158.195
C00679=1026.699,-125.836,-85.588,166.570,44.866,158.195
C00680=1026.705,-125.587,-85.596,166.572,44.863,158.195
C00681=1026.710,-125.337,-85.604,166.575,44.860,158.195
C00682=1026.716,-125.088,-85.612,166.578,44.857,158.195
C00683=1026.721,-124.838,-85.621,166.581,44.855,158.195
C00684=1026.728,-124.588,-85.629,166.584,44.852,158.195
C00685=1026.733,-124.338,-85.638,166.587,44.849,158.194
C00686=1026.738,-124.088,-85.646,166.590,44.847,158.194
C00687=1026.744,-123.838,-85.655,166.593,44.845,158.194
C00688=1026.750,-123.588,-85.663,166.596,44.842,158.194
C00689=1026.755,-123.339,-85.671,166.599,44.839,158.194
C00690=1026.761,-123.089,-85.680,166.602,44.837,158.194
C00691=1026.767,-122.839,-85.688,166.605,44.834,158.193
C00692=1026.772,-122.589,-85.697,166.607,44.831,158.193
C00693=1026.778,-122.339,-85.705,166.611,44.829,158.193
C00694=1026.783,-122.090,-85.714,166.613,44.827,158.193
C00695=1026.790,-121.840,-85.722,166.617,44.824,158.193
C00696=1026.795,-121.590,-85.730,166.619,44.822,158.193
C00697=1026.800,-121.340,-85.739,166.623,44.819,158.193
C00698=1026.807,-121.091,-85.748,166.625,44.816,158.192
C00699=1026.812,-120.841,-85.756,166.629,44.814,158.192
C00700=1026.818,-120.591,-85.765,166.631,44.811,158.192
C00701=1026.823,-120.341,-85.774,166.635,44.809,158.192
C00702=1026.829,-120.091,-85.781,166.637,44.806,158.192
C00703=1026.835,-119.842,-85.790,166.640,44.803,158.192
C00704=1026.841,-119.591,-85.799,166.643,44.801,158.192
C00705=1026.846,-119.342,-85.808,166.646,44.799,158.192
C00706=1026.852,-119.093,-85.816,166.649,44.796,158.191
C00707=1026.858,-118.842,-85.825,166.652,44.794,158.191
C00708=1026.863,-118.593,-85.833,166.655,44.791,158.191
C00709=1026.869,-118.343,-85.842,166.658,44.788,158.191
C00710=1026.874,-118.093,-85.851,166.661,44.786,158.191
C00711=1026.881,-117.844,-85.859,166.664,44.783,158.191
C00712=1026.887,-117.593,-85.868,166.667,44.781,158.190
C00713=1026.893,-117.308,-85.878,166.670,44.778,158.190
C00714=1026.899,-117.021,-85.888,166.673,44.775,158.190
C00715=1026.906,-116.736,-85.898,166.677,44.772,158.190
C00716=1026.912,-116.450,-85.908,166.680,44.769,158.190
C00717=1026.918,-116.200,-85.916,166.684,44.767,158.190
C00718=1026.924,-115.950,-85.925,166.686,44.764,158.190
C00719=1026.930,-115.701,-85.934,166.690,44.762,158.190
C00720=1026.935,-115.450,-85.943,166.692,44.759,158.189
C00721=1026.941,-115.201,-85.951,166.696,44.756,158.189
C00722=1026.947,-114.951,-85.961,166.698,44.754,158.189
C00723=1026.953,-114.702,-85.969,166.702,44.752,158.189
C00724=1026.959,-114.451,-85.978,166.704,44.750,158.189
C00725=1026.964,-114.202,-85.987,166.708,44.747,158.189
C00726=1026.970,-113.952,-85.996,166.710,44.744,158.188
C00727=1026.976,-113.703,-86.005,166.714,44.742,158.188
C00728=1026.981,-113.453,-86.013,166.716,44.739,158.188
C00729=1026.987,-113.202,-86.022,166.720,44.737,158.188
C00730=1026.993,-112.953,-86.031,166.722,44.734,158.188
C00731=1026.998,-112.703,-86.040,166.726,44.732,158.188
C00732=1027.004,-112.454,-86.050,166.728,44.729,158.188
C00733=1027.010,-112.203,-86.058,166.732,44.727,158.188
C00734=1027.015,-111.954,-86.068,166.734,44.725,158.187
C00735=1027.021,-111.704,-86.076,166.738,44.722,158.187
C00736=1027.027,-111.455,-86.086,166.740,44.720,158.187
C00737=1027.033,-111.204,-86.094,166.743,44.717,158.187
C00738=1027.039,-110.955,-86.104,166.746,44.715,158.187
C00739=1027.044,-110.705,-86.113,166.749,44.712,158.187
C00740=1027.050,-110.455,-86.122,166.752,44.710,158.187
C00741=1027.056,-110.205,-86.131,166.754,44.707,158.186
C00742=1027.062,-109.955,-86.140,166.758,44.705,158.186
C00743=1027.067,-109.706,-86.149,166.760,44.702,158.186
C00744=1027.074,-109.456,-86.158,166.764,44.700,158.186
C00745=1027.079,-109.207,-86.166,166.766,44.698,158.186
C00746=1027.085,-108.957,-86.176,166.770,44.695,158.186
C00747=1027.091,-108.706,-86.185,166.772,44.693,158.186
C00748=1027.097,-108.457,-86.194,166.776,44.690,158.186
C00749=1027.103,-108.207,-86.203,166.778,44.688,158.185
C00750=1027.108,-107.958,-86.212,166.782,44.685,158.185
C00751=1027.114,-107.708,-86.221,166.785,44.683,158.185
C00752=1027.121,-107.458,-86.231,166.788,44.680,158.185
C00753=1027.125,-107.208,-86.240,166.791,44.678,158.185
C00754=1027.131,-106.958,-86.250,166.794,44.675,158.185
C00755=1027.137,-106.709,-86.259,166.797,44.673,158.185
C00756=1027.143,-106.459,-86.268,166.799,44.671,158.184
C00757=1027.149,-106.209,-86.277,166.803,44.668,158.184
C00758=1027.154,-105.960,-86.286,166.805,44.666,158.184
C00759=1027.160,-105.709,-86.295,166.809,44.664,158.184
C00760=1027.166,-105.460,-86.305,166.811,44.662,158.184
C00761=1027.171,-105.210,-86.315,166.815,44.659,158.184
C00762=1027.177,-104.960,-86.324,166.817,44.657,158.184
C00763=1027.183,-104.711,-86.333,166.821,44.654,158.184
C00764=1027.189,-104.461,-86.342,166.823,44.652,158.184
C00765=1027.195,-104.211,-86.352,166.826,44.649,158.183
C00766=1027.201,-103.962,-86.361,166.829,44.647,158.183
C00767=1027.207,-103.712,-86.370,166.832,44.644,158.183
C00768=1027.212,-103.462,-86.380,166.835,44.642,158.183
C00769=1027.218,-103.212,-86.389,166.838,44.640,158.183
C00770=1027.224,-102.963,-86.399,166.841,44.637,158.183
C00771=1027.230,-102.713,-86.408,166.844,44.635,158.183
C00772=1027.236,-102.463,-86.418,166.847,44.633,158.183
C00773=1027.241,-102.213,-86.427,166.850,44.631,158.182
C00774=1027.247,-101.963,-86.437,166.852,44.628,158.182
C00775=1027.253,-101.713,-86.446,166.856,44.626,158.182
C00776=1027.258,-101.464,-86.455,166.858,44.624,158.182
C00777=1027.265,-101.178,-86.466,166.862,44.621,158.182
C00778=1027.272,-100.891,-86.477,166.865,44.618,158.182
C00779=1027.279,-100.605,-86.489,166.869,44.615,158.182
C00780=1027.286,-100.319,-86.499,166.872,44.612,158.181
C00781=1027.292,-100.069,-86.509,166.875,44.610,158.181
C00782=1027.297,-99.820,-86.518,166.878,44.608,158.181
C00783=1027.303,-99.570,-86.528,166.881,44.606,158.181
C00784=1027.309,-99.320,-86.538,166.884,44.603,158.181
C00785=1027.315,-99.070,-86.548,166.887,44.601,158.181
C00786=1027.321,-98.820,-86.556,166.890,44.599,158.181
C00787=1027.326,-98.570,-86.566,166.893,44.596,158.181
C00788=1027.332,-98.320,-86.576,166.896,44.594,158.181
C00789=1027.338,-98.071,-86.585,166.899,44.591,158.180
C00790=1027.344,-97.821,-86.595,166.901,44.589,158.180
C00791=1027.350,-97.571,-86.605,166.905,44.587,158.180
C00792=1027.356,-97.322,-86.615,166.907,44.584,158.180
C00793=1027.361,-97.072,-86.625,166.911,44.582,158.180
C00794=1027.367,-96.822,-86.635,166.914,44.580,158.180
C00795=1027.373,-96.572,-86.644,166.916,44.578,158.180
C00796=1027.379,-96.322,-86.654,166.920,44.575,158.180
C00797=1027.384,-96.073,-86.664,166.922,44.573,158.179
C00798=1027.390,-95.823,-86.674,166.925,44.571,158.179
C00799=1027.396,-95.573,-86.683,166.928,44.568,158.179
C00800=1027.402,-95.324,-86.694,166.931,44.567,158.179
C00801=1027.408,-95.074,-86.704,166.934,44.564,158.179
C00802=1027.413,-94.824,-86.714,166.937,44.562,158.179
C00803=1027.419,-94.575,-86.723,166.939,44.560,158.179
C00804=1027.424,-94.325,-86.733,166.943,44.558,158.179
C00805=1027.431,-94.076,-86.744,166.946,44.556,158.179
C00806=1027.436,-93.825,-86.754,166.948,44.554,158.179
C00807=1027.442,-93.576,-86.763,166.952,44.551,158.178
C00808=1027.448,-93.326,-86.774,166.954,44.549,158.178
C00809=1027.454,-93.076,-86.783,166.957,44.547,158.178
C00810=1027.460,-92.826,-86.794,166.961,44.545,158.178
C00811=1027.465,-92.577,-86.803,166.963,44.542,158.178
C00812=1027.471,-92.327,-86.813,166.967,44.540,158.178
C00813=1027.477,-92.078,-86.824,166.969,44.538,158.178
C00814=1027.483,-91.828,-86.834,166.972,44.535,158.178
C00815=1027.489,-91.578,-86.843,166.975,44.533,158.178
C00816=1027.494,-91.328,-86.853,166.978,44.531,158.177
C00817=1027.501,-91.079,-86.864,166.980,44.529,158.177
C00818=1027.506,-90.829,-86.874,166.984,44.526,158.177
C00819=1027.512,-90.579,-86.884,166.986,44.524,158.177
C00820=1027.518,-90.329,-86.894,166.990,44.522,158.177
C00821=1027.524,-90.079,-86.904,166.992,44.520,158.177
C00822=1027.530,-89.829,-86.914,166.995,44.518,158.177
C00823=1027.536,-89.580,-86.924,166.999,44.515,158.177
C00824=1027.542,-89.330,-86.935,167.001,44.513,158.177
C00825=1027.548,-89.080,-86.944,167.004,44.511,158.176
C00826=1027.554,-88.831,-86.955,167.007,44.509,158.176
C00827=1027.559,-88.581,-86.965,167.010,44.507,158.176
C00828=1027.565,-88.331,-86.975,167.013,44.504,158.176
C00829=1027.571,-88.081,-86.986,167.016,44.502,158.176
C00830=1027.577,-87.832,-86.995,167.019,44.500,158.176
C00831=1027.583,-87.582,-87.006,167.022,44.498,158.176
C00832=1027.589,-87.332,-87.016,167.025,44.495,158.176
C00833=1027.595,-87.083,-87.026,167.027,44.493,158.175
C00834=1027.601,-86.833,-87.036,167.031,44.491,158.175
C00835=1027.607,-86.584,-87.047,167.033,44.488,158.175
C00836=1027.613,-86.334,-87.057,167.037,44.486,158.175
C00837=1027.619,-86.084,-87.067,167.039,44.484,158.175
C00838=1027.625,-85.834,-87.077,167.042,44.482,158.175
C00839=1027.630,-85.585,-87.088,167.045,44.479,158.175
C00840=1027.636,-85.335,-87.098,167.048,44.477,158.175
C00841=1027.643,-85.051,-87.109,167.052,44.475,158.175
C00842=1027.650,-84.766,-87.121,167.055,44.472,158.174
C00843=1027.657,-84.483,-87.134,167.059,44.470,158.174
C00844=1027.664,-84.198,-87.145,167.061,44.467,158.174
C00845=1027.669,-83.948,-87.155,167.065,44.465,158.174
C00846=1027.676,-83.699,-87.165,167.067,44.463,158.174
C00847=1027.681,-83.449,-87.175,167.071,44.460,158.174
C00848=1027.688,-83.200,-87.186,167.073,44.458,158.174
C00849=1027.694,-82.950,-87.197,167.076,44.456,158.174
C00850=1027.700,-82.699,-87.207,167.079,44.453,158.173
C00851=1027.706,-82.450,-87.217,167.082,44.451,158.173
C00852=1027.712,-82.200,-87.228,167.084,44.449,158.173
C00853=1027.718,-81.951,-87.238,167.088,44.446,158.173
C00854=1027.724,-81.701,-87.249,167.090,44.445,158.173
C00855=1027.730,-81.452,-87.258,167.094,44.442,158.173
C00856=1027.736,-81.201,-87.270,167.096,44.440,158.173
C00857=1027.742,-80.952,-87.280,167.099,44.438,158.173
C00858=1027.748,-80.702,-87.290,167.103,44.436,158.173
C00859=1027.754,-80.453,-87.301,167.105,44.434,158.172
C00860=1027.760,-80.203,-87.311,167.108,44.431,158.172
C00861=1027.766,-79.953,-87.322,167.111,44.429,158.172
C00862=1027.772,-79.703,-87.333,167.114,44.427,158.172
C00863=1027.778,-79.454,-87.343,167.117,44.425,158.172
C00864=1027.783,-79.204,-87.354,167.120,44.422,158.172
C00865=1027.790,-78.954,-87.364,167.123,44.420,158.172
C00866=1027.796,-78.704,-87.375,167.125,44.418,158.172
C00867=1027.802,-78.455,-87.386,167.129,44.416,158.172
C00868=1027.808,-78.205,-87.397,167.131,44.414,158.171
C00869=1027.813,-77.956,-87.408,167.134,44.412,158.171
C00870=1027.819,-77.706,-87.418,167.138,44.410,158.171
C00871=1027.826,-77.456,-87.429,167.140,44.407,158.171
C00872=1027.832,-77.206,-87.439,167.143,44.405,158.171
C00873=1027.837,-76.957,-87.450,167.145,44.403,158.171
C00874=1027.843,-76.707,-87.461,167.149,44.401,158.171
C00875=1027.849,-76.457,-87.472,167.152,44.399,158.171
C00876=1027.855,-76.208,-87.483,167.154,44.397,158.171
C00877=1027.861,-75.958,-87.493,167.158,44.395,158.170
C00878=1027.867,-75.708,-87.504,167.160,44.393,158.170
C00879=1027.873,-75.458,-87.515,167.163,44.391,158.170
C00880=1027.879,-75.209,-87.526,167.166,44.389,158.170
C00881=1027.885,-74.959,-87.537,167.169,44.387,158.170
C00882=1027.891,-74.709,-87.548,167.172,44.385,158.170
C00883=1027.897,-74.459,-87.559,167.175,44.382,158.170
C00884=1027.903,-74.210,-87.569,167.178,44.380,158.170
C00885=1027.908,-73.960,-87.581,167.180,44.378,158.170
C00886=1027.915,-73.710,-87.592,167.183,44.376,158.170
C00887=1027.921,-73.461,-87.603,167.187,44.374,158.169
C00888=1027.926,-73.211,-87.614,167.189,44.372,158.169
C00889=1027.933,-72.961,-87.625,167.192,44.370,158.169
C00890=1027.938,-72.712,-87.636,167.194,44.368,158.169
C00891=1027.944,-72.462,-87.647,167.197,44.366,158.169
C00892=1027.950,-72.212,-87.659,167.201,44.364,158.169
C00893=1027.956,-71.963,-87.670,167.203,44.362,158.169
C00894=1027.961,-71.713,-87.681,167.206,44.360,158.169
C00895=1027.967,-71.464,-87.692,167.208,44.358,158.169
C00896=1027.974,-71.214,-87.703,167.212,44.356,158.169
C00897=1027.979,-70.964,-87.714,167.215,44.354,158.169
C00898=1027.985,-70.715,-87.725,167.217,44.352,158.168
C00899=1027.991,-70.464,-87.737,167.220,44.350,158.168
C00900=1027.997,-70.215,-87.748,167.224,44.348,158.168
C00901=1028.003,-69.965,-87.760,167.226,44.346,158.168
C00902=1028.009,-69.716,-87.770,167.229,44.344,158.168
///RCONF 1,0,0,1,0,0,0,0,0,0,0,0,0,0,0,0,0,0,0,0,0,0,0,0
C00903=1028.015,-69.466,-87.781,167.231,44.342,158.168
C00904=1028.021,-69.216,-87.793,167.234,44.340,158.168
C00905=1028.027,-68.935,-87.806,167.238,44.338,158.168
C00906=1028.033,-68.653,-87.819,167.241,44.336,158.168
C00907=1028.041,-68.370,-87.831,167.244,44.334,158.168
C00908=1028.047,-68.088,-87.844,167.247,44.331,158.168
C00909=1028.053,-67.838,-87.855,167.250,44.329,158.167
C00910=1028.059,-67.589,-87.866,167.254,44.327,158.167
C00911=1028.065,-67.340,-87.877,167.256,44.325,158.167
C00912=1028.071,-67.089,-87.889,167.259,44.323,158.167
C00913=1028.077,-66.840,-87.901,167.261,44.321,158.167
C00914=1028.083,-66.590,-87.912,167.264,44.319,158.167
C00915=1028.089,-66.341,-87.923,167.268,44.317,158.167
C00916=1028.095,-66.090,-87.934,167.270,44.315,158.167
C00917=1028.101,-65.842,-87.946,167.273,44.313,158.167
C00918=1028.107,-65.591,-87.957,167.276,44.311,158.167
C00919=1028.113,-65.342,-87.968,167.279,44.309,158.167
C00920=1028.119,-65.093,-87.980,167.282,44.307,158.167
C00921=1028.125,-64.843,-87.991,167.284,44.305,158.166
C00922=1028.131,-64.593,-88.002,167.287,44.303,158.166
C00923=1028.137,-64.343,-88.015,167.290,44.301,158.166
C00924=1028.142,-64.094,-88.026,167.293,44.299,158.166
C00925=1028.149,-63.844,-88.037,167.296,44.297,158.166
C00926=1028.155,-63.595,-88.048,167.299,44.295,158.166
C00927=1028.161,-63.344,-88.060,167.301,44.293,158.166
C00928=1028.166,-63.095,-88.072,167.305,44.291,158.166
C00929=1028.173,-62.845,-88.083,167.307,44.289,158.166
C00930=1028.179,-62.596,-88.095,167.310,44.287,158.166
C00931=1028.185,-62.346,-88.106,167.313,44.285,158.165
C00932=1028.192,-62.096,-88.117,167.316,44.283,158.165
C00933=1028.197,-61.847,-88.129,167.319,44.281,158.165
C00934=1028.203,-61.596,-88.141,167.321,44.279,158.165
C00935=1028.209,-61.348,-88.152,167.324,44.277,158.165
C00936=1028.216,-61.097,-88.163,167.326,44.275,158.165
C00937=1028.222,-60.848,-88.175,167.330,44.273,158.165
C00938=1028.227,-60.598,-88.187,167.333,44.271,158.165
C00939=1028.233,-60.349,-88.198,167.335,44.269,158.165
C00940=1028.240,-60.099,-88.210,167.338,44.267,158.165
C00941=1028.246,-59.849,-88.222,167.342,44.265,158.164
C00942=1028.252,-59.600,-88.232,167.344,44.263,158.164
C00943=1028.258,-59.350,-88.245,167.347,44.261,158.164
C00944=1028.264,-59.100,-88.256,167.349,44.259,158.164
C00945=1028.270,-58.851,-88.268,167.352,44.257,158.164
C00946=1028.277,-58.601,-88.279,167.356,44.255,158.164
C00947=1028.283,-58.352,-88.291,167.358,44.253,158.164
C00948=1028.289,-58.102,-88.303,167.361,44.251,158.164
C00949=1028.295,-57.852,-88.314,167.364,44.249,158.164
C00950=1028.301,-57.603,-88.326,167.367,44.247,158.164
C00951=1028.307,-57.353,-88.337,167.370,44.244,158.163
C00952=1028.313,-57.103,-88.350,167.372,44.242,158.163
C00953=1028.319,-56.854,-88.361,167.375,44.240,158.163
C00954=1028.326,-56.604,-88.373,167.377,44.238,158.163
C00955=1028.332,-56.354,-88.385,167.381,44.236,158.163
C00956=1028.337,-56.104,-88.396,167.384,44.234,158.163
C00957=1028.344,-55.855,-88.408,167.386,44.232,158.163
C00958=1028.351,-55.605,-88.420,167.389,44.231,158.163
C00959=1028.356,-55.356,-88.431,167.393,44.228,158.163
C00960=1028.362,-55.106,-88.444,167.395,44.227,158.163
C00961=1028.369,-54.856,-88.455,167.398,44.225,158.162
C00962=1028.375,-54.607,-88.466,167.400,44.222,158.162
C00963=1028.381,-54.357,-88.478,167.403,44.220,158.162
C00964=1028.387,-54.107,-88.491,167.406,44.218,158.162
C00965=1028.394,-53.858,-88.503,167.409,44.216,158.162
C00966=1028.399,-53.608,-88.514,167.412,44.214,158.162
C00967=1028.406,-53.359,-88.526,167.414,44.212,158.162
C00968=1028.412,-53.109,-88.538,167.418,44.210,158.162
C00969=1028.419,-52.828,-88.551,167.420,44.207,158.161
C00970=1028.427,-52.547,-88.564,167.424,44.205,158.161
C00971=1028.433,-52.266,-88.578,167.427,44.203,158.161
C00972=1028.441,-51.986,-88.591,167.430,44.200,158.161
C00973=1028.449,-51.634,-88.608,167.434,44.197,158.161
C00974=1028.458,-51.282,-88.624,167.438,44.195,158.161
C00975=1028.464,-51.032,-88.636,167.440,44.193,158.161
C00976=1028.470,-50.783,-88.648,167.443,44.191,158.161
C00977=1028.477,-50.533,-88.660,167.447,44.189,158.160
C00978=1028.483,-50.283,-88.673,167.449,44.187,158.160
C00979=1028.488,-50.034,-88.685,167.452,44.185,158.160
C00980=1028.495,-49.784,-88.697,167.454,44.183,158.160
C00981=1028.501,-49.534,-88.710,167.457,44.182,158.160
C00982=1028.507,-49.285,-88.722,167.460,44.180,158.160
C00983=1028.513,-49.035,-88.734,167.463,44.178,158.160
C00984=1028.519,-48.786,-88.746,167.465,44.176,158.160
C00985=1028.525,-48.536,-88.758,167.469,44.174,158.160
C00986=1028.531,-48.286,-88.771,167.471,44.172,158.160
C00987=1028.537,-48.036,-88.783,167.474,44.170,158.160
C00988=1028.544,-47.787,-88.795,167.477,44.168,158.159
C00989=1028.549,-47.538,-88.807,167.480,44.167,158.159
C00990=1028.555,-47.288,-88.820,167.482,44.165,158.159
C00991=1028.561,-47.038,-88.832,167.485,44.163,158.159
C00992=1028.567,-46.788,-88.845,167.487,44.161,158.159
C00993=1028.573,-46.538,-88.857,167.491,44.159,158.159
C00994=1028.579,-46.290,-88.869,167.494,44.157,158.159
C00995=1028.585,-46.040,-88.881,167.496,44.155,158.159
C00996=1028.591,-45.790,-88.894,167.499,44.153,158.159
C00997=1028.598,-45.540,-88.906,167.501,44.151,158.159
C00998=1028.604,-45.290,-88.918,167.504,44.149,158.159
C00999=1028.610,-45.040,-88.931,167.507,44.147,158.158
C01000=1028.617,-44.792,-88.944,167.510,44.146,158.158
C01001=1028.622,-44.542,-88.956,167.512,44.144,158.158
C01002=1028.628,-44.292,-88.968,167.516,44.142,158.158
C01003=1028.634,-44.043,-88.980,167.518,44.140,158.158
C01004=1028.640,-43.793,-88.993,167.521,44.138,158.158
C01005=1028.646,-43.543,-89.005,167.524,44.136,158.158
C01006=1028.653,-43.294,-89.017,167.526,44.134,158.158
C01007=1028.659,-43.044,-89.031,167.529,44.132,158.158
C01008=1028.665,-42.794,-89.043,167.531,44.130,158.158
C01009=1028.672,-42.545,-89.055,167.534,44.128,158.158
C01010=1028.678,-42.295,-89.068,167.537,44.127,158.157
C01011=1028.683,-42.045,-89.080,167.540,44.124,158.157
C01012=1028.690,-41.796,-89.093,167.543,44.122,158.157
C01013=1028.696,-41.546,-89.105,167.546,44.121,158.157
C01014=1028.702,-41.297,-89.118,167.548,44.119,158.157
C01015=1028.708,-41.048,-89.130,167.551,44.117,158.157
C01016=1028.715,-40.798,-89.143,167.554,44.115,158.157
C01017=1028.720,-40.548,-89.155,167.556,44.114,158.157
C01018=1028.727,-40.299,-89.167,167.559,44.112,158.157
C01019=1028.733,-40.049,-89.180,167.562,44.110,158.157
C01020=1028.739,-39.800,-89.193,167.565,44.108,158.157
C01021=1028.746,-39.550,-89.205,167.568,44.106,158.156
C01022=1028.752,-39.300,-89.218,167.570,44.104,158.156
C01023=1028.758,-39.051,-89.231,167.573,44.102,158.156
C01024=1028.764,-38.801,-89.244,167.576,44.100,158.156
C01025=1028.770,-38.551,-89.256,167.578,44.098,158.156
C01026=1028.776,-38.302,-89.269,167.581,44.097,158.156
C01027=1028.782,-38.052,-89.282,167.584,44.095,158.156
C01028=1028.788,-37.802,-89.294,167.586,44.093,158.156
C01029=1028.795,-37.553,-89.307,167.589,44.091,158.156
C01030=1028.801,-37.303,-89.320,167.592,44.089,158.156
C01031=1028.809,-36.949,-89.339,167.595,44.087,158.156
C01032=1028.818,-36.595,-89.356,167.600,44.084,158.155
C01033=1028.827,-36.241,-89.375,167.603,44.082,158.155
C01034=1028.836,-35.887,-89.393,167.607,44.079,158.155
C01035=1028.842,-35.637,-89.406,167.609,44.077,158.155
C01036=1028.848,-35.387,-89.419,167.613,44.075,158.155
C01037=1028.854,-35.138,-89.432,167.616,44.074,158.155
C01038=1028.860,-34.888,-89.444,167.618,44.072,158.155
C01039=1028.866,-34.639,-89.458,167.621,44.070,158.155
C01040=1028.872,-34.389,-89.470,167.624,44.068,158.155
C01041=1028.878,-34.140,-89.483,167.626,44.066,158.155
///RCONF 1,0,0,0,0,0,0,0,0,0,0,0,0,0,0,0,0,0,0,0,0,0,0,0
C01042=1028.884,-33.890,-89.496,167.629,44.064,158.154
C01043=1028.890,-33.641,-89.509,167.632,44.063,158.154
C01044=1028.897,-33.391,-89.523,167.634,44.061,158.154
C01045=1028.903,-33.141,-89.535,167.637,44.059,158.154
C01046=1028.909,-32.892,-89.549,167.640,44.057,158.154
C01047=1028.915,-32.642,-89.561,167.642,44.055,158.154
C01048=1028.921,-32.392,-89.575,167.645,44.053,158.154
C01049=1028.927,-32.143,-89.587,167.647,44.051,158.154
C01050=1028.933,-31.893,-89.600,167.650,44.050,158.154
C01051=1028.940,-31.644,-89.614,167.653,44.048,158.154
C01052=1028.946,-31.394,-89.626,167.655,44.046,158.154
C01053=1028.952,-31.144,-89.640,167.658,44.044,158.153
C01054=1028.959,-30.895,-89.653,167.661,44.043,158.153
C01055=1028.964,-30.645,-89.666,167.663,44.041,158.153
C01056=1028.971,-30.396,-89.679,167.666,44.039,158.153
C01057=1028.977,-30.147,-89.692,167.669,44.037,158.153
C01058=1028.983,-29.897,-89.705,167.671,44.036,158.153
C01059=1028.989,-29.647,-89.718,167.674,44.034,158.153
C01060=1028.996,-29.397,-89.732,167.677,44.032,158.153
C01061=1029.002,-29.148,-89.744,167.679,44.030,158.153
C01062=1029.008,-28.898,-89.757,167.683,44.028,158.153
C01063=1029.014,-28.649,-89.771,167.686,44.026,158.153
C01064=1029.020,-28.399,-89.783,167.688,44.024,158.152
C01065=1029.027,-28.149,-89.797,167.691,44.022,158.152
C01066=1029.033,-27.900,-89.810,167.693,44.020,158.152
C01067=1029.039,-27.651,-89.823,167.696,44.019,158.152
C01068=1029.045,-27.401,-89.836,167.699,44.017,158.152
C01069=1029.051,-27.151,-89.849,167.701,44.015,158.152
C01070=1029.058,-26.902,-89.863,167.704,44.013,158.152
C01071=1029.064,-26.652,-89.876,167.707,44.011,158.152
C01072=1029.071,-26.403,-89.889,167.710,44.010,158.152
C01073=1029.076,-26.153,-89.903,167.712,44.008,158.152
C01074=1029.082,-25.904,-89.916,167.715,44.006,158.152
C01075=1029.089,-25.654,-89.930,167.717,44.004,158.151
C01076=1029.095,-25.404,-89.943,167.719,44.003,158.151
C01077=1029.101,-25.155,-89.957,167.722,44.001,158.151
C01078=1029.107,-24.905,-89.970,167.724,43.999,158.151
C01079=1029.114,-24.655,-89.984,167.727,43.997,158.151
C01080=1029.120,-24.406,-89.997,167.730,43.996,158.151
C01081=1029.125,-24.157,-90.011,167.733,43.994,158.151
C01082=1029.132,-23.907,-90.024,167.735,43.992,158.151
C01083=1029.138,-23.657,-90.037,167.738,43.990,158.151
C01084=1029.143,-23.407,-90.051,167.741,43.989,158.151
C01085=1029.150,-23.158,-90.064,167.743,43.987,158.151
C01086=1029.156,-22.909,-90.077,167.746,43.985,158.150
C01087=1029.163,-22.659,-90.091,167.748,43.983,158.150
C01088=1029.168,-22.409,-90.105,167.751,43.982,158.150
C01089=1029.174,-22.160,-90.118,167.754,43.980,158.150
C01090=1029.181,-21.910,-90.132,167.757,43.978,158.150
C01091=1029.187,-21.661,-90.145,167.759,43.976,158.150
C01092=1029.193,-21.411,-90.159,167.762,43.975,158.150
C01093=1029.199,-21.162,-90.172,167.765,43.973,158.150
C01094=1029.206,-20.912,-90.186,167.767,43.971,158.150
C01095=1029.213,-20.631,-90.201,167.770,43.969,158.150
C01096=1029.220,-20.350,-90.217,167.773,43.967,158.150
C01097=1029.227,-20.068,-90.232,167.776,43.965,158.150
C01098=1029.234,-19.787,-90.247,167.779,43.964,158.149
C01099=1029.240,-19.538,-90.261,167.781,43.962,158.149
C01100=1029.246,-19.288,-90.275,167.784,43.960,158.149
C01101=1029.253,-19.038,-90.288,167.787,43.958,158.149
C01102=1029.259,-18.789,-90.301,167.789,43.956,158.149
C01103=1029.264,-18.539,-90.315,167.792,43.955,158.149
C01104=1029.271,-18.290,-90.329,167.795,43.953,158.149
C01105=1029.277,-18.040,-90.342,167.797,43.951,158.149
C01106=1029.284,-17.791,-90.357,167.800,43.949,158.149
C01107=1029.290,-17.541,-90.370,167.803,43.947,158.148
C01108=1029.296,-17.292,-90.384,167.805,43.945,158.148
C01109=1029.303,-17.042,-90.397,167.808,43.944,158.148
C01110=1029.308,-16.793,-90.411,167.811,43.942,158.148
C01111=1029.315,-16.543,-90.425,167.813,43.940,158.148
C01112=1029.321,-16.293,-90.438,167.816,43.938,158.148
C01113=1029.327,-16.044,-90.453,167.818,43.936,158.148
C01114=1029.334,-15.794,-90.466,167.821,43.934,158.148
C01115=1029.340,-15.545,-90.480,167.824,43.933,158.148
C01116=1029.346,-15.295,-90.494,167.825,43.931,158.148
C01117=1029.353,-15.046,-90.507,167.828,43.930,158.148
C01118=1029.359,-14.796,-90.522,167.831,43.928,158.148
C01119=1029.364,-14.546,-90.536,167.834,43.926,158.147
C01120=1029.371,-14.297,-90.549,167.836,43.924,158.147
C01121=1029.377,-14.047,-90.564,167.839,43.923,158.147
C01122=1029.383,-13.798,-90.577,167.842,43.921,158.147
C01123=1029.389,-13.548,-90.592,167.844,43.919,158.147
C01124=1029.396,-13.299,-90.606,167.847,43.918,158.147
C01125=1029.401,-13.050,-90.619,167.850,43.916,158.147
C01126=1029.408,-12.800,-90.633,167.851,43.915,158.147
C01127=1029.414,-12.551,-90.648,167.854,43.913,158.147
C01128=1029.420,-12.300,-90.662,167.857,43.911,158.147
C01129=1029.426,-12.051,-90.675,167.859,43.910,158.147
C01130=1029.433,-11.802,-90.690,167.862,43.908,158.146
C01131=1029.439,-11.552,-90.703,167.865,43.906,158.146
C01132=1029.445,-11.303,-90.718,167.867,43.904,158.146
C01133=1029.451,-11.053,-90.732,167.870,43.903,158.146
C01134=1029.457,-10.803,-90.746,167.873,43.901,158.146
C01135=1029.463,-10.554,-90.760,167.874,43.899,158.146
C01136=1029.470,-10.304,-90.774,167.877,43.898,158.146
C01137=1029.476,-10.055,-90.789,167.880,43.896,158.146
C01138=1029.483,-9.805,-90.802,167.882,43.894,158.146
C01139=1029.488,-9.556,-90.817,167.885,43.892,158.146
C01140=1029.495,-9.306,-90.830,167.888,43.891,158.146
C01141=1029.501,-9.057,-90.844,167.890,43.889,158.146
C01142=1029.507,-8.807,-90.859,167.893,43.887,158.145
C01143=1029.513,-8.558,-90.873,167.896,43.885,158.145
C01144=1029.520,-8.308,-90.887,167.898,43.884,158.145
C01145=1029.526,-8.059,-90.901,167.900,43.882,158.145
C01146=1029.532,-7.809,-90.916,167.903,43.880,158.145
C01147=1029.538,-7.560,-90.930,167.905,43.878,158.145
C01148=1029.545,-7.310,-90.944,167.908,43.877,158.145
C01149=1029.551,-7.060,-90.958,167.911,43.875,158.145
C01150=1029.558,-6.811,-90.972,167.913,43.873,158.145
C01151=1029.564,-6.561,-90.986,167.916,43.871,158.145
C01152=1029.569,-6.312,-91.001,167.919,43.870,158.145
C01153=1029.576,-6.063,-91.015,167.921,43.868,158.144
C01154=1029.582,-5.813,-91.029,167.923,43.867,158.144
C01155=1029.589,-5.564,-91.044,167.926,43.865,158.144
C01156=1029.595,-5.314,-91.058,167.928,43.863,158.144
C01157=1029.601,-5.065,-91.072,167.931,43.862,158.144
C01158=1029.608,-4.815,-91.086,167.934,43.860,158.144
C01159=1029.615,-4.533,-91.103,167.936,43.858,158.144
C01160=1029.622,-4.249,-91.118,167.939,43.856,158.144
C01161=1029.629,-3.967,-91.134,167.943,43.854,158.144
C01162=1029.636,-3.684,-91.151,167.945,43.852,158.143
C01163=1029.642,-3.433,-91.166,167.948,43.850,158.143
C01164=1029.648,-3.185,-91.180,167.951,43.849,158.143
C01165=1029.654,-2.935,-91.195,167.952,43.847,158.143
C01166=1029.660,-2.686,-91.210,167.955,43.845,158.143
C01167=1029.666,-2.436,-91.224,167.958,43.844,158.143
C01168=1029.673,-2.186,-91.239,167.961,43.842,158.143
C01169=1029.678,-1.937,-91.254,167.963,43.841,158.143
C01170=1029.685,-1.687,-91.269,167.965,43.839,158.143
C01171=1029.691,-1.439,-91.282,167.968,43.837,158.143
C01172=1029.697,-1.188,-91.297,167.970,43.836,158.143
C01173=1029.704,-0.939,-91.312,167.973,43.834,158.143
C01174=1029.710,-0.690,-91.326,167.976,43.833,158.143
C01175=1029.716,-0.440,-91.341,167.977,43.831,158.142
C01176=1029.722,-0.191,-91.356,167.980,43.829,158.142
C01177=1029.728,0.059,-91.370,167.983,43.828,158.142
C01178=1029.734,0.309,-91.385,167.986,43.826,158.142
C01179=1029.740,0.558,-91.400,167.988,43.825,158.142
C01180=1029.746,0.807,-91.414,167.990,43.823,158.142
C01181=1029.753,1.057,-91.429,167.993,43.821,158.142
C01182=1029.759,1.306,-91.444,167.995,43.820,158.142
C01183=1029.765,1.556,-91.459,167.998,43.818,158.142
C01184=1029.771,1.805,-91.474,168.001,43.816,158.142
C01185=1029.777,2.056,-91.488,168.003,43.815,158.142
C01186=1029.783,2.304,-91.503,168.005,43.813,158.142
C01187=1029.790,2.554,-91.518,168.008,43.811,158.141
C01188=1029.796,2.804,-91.533,168.011,43.810,158.141
C01189=1029.802,3.053,-91.547,168.013,43.808,158.141
C01190=1029.808,3.302,-91.562,168.015,43.807,158.141
C01191=1029.815,3.552,-91.577,168.018,43.805,158.141
C01192=1029.820,3.801,-91.592,168.020,43.804,158.141
C01193=1029.827,4.051,-91.607,168.023,43.802,158.141
C01194=1029.833,4.300,-91.622,168.026,43.800,158.141
C01195=1029.839,4.550,-91.636,168.027,43.799,158.141
C01196=1029.846,4.799,-91.650,168.030,43.797,158.141
C01197=1029.852,5.048,-91.665,168.033,43.796,158.141
C01198=1029.859,5.298,-91.680,168.035,43.794,158.140
C01199=1029.865,5.548,-91.695,168.038,43.792,158.140
C01200=1029.871,5.797,-91.710,168.040,43.791,158.140
C01201=1029.877,6.046,-91.725,168.042,43.789,158.140
C01202=1029.884,6.296,-91.740,168.045,43.787,158.140
C01203=1029.890,6.546,-91.755,168.048,43.786,158.140
C01204=1029.896,6.795,-91.770,168.051,43.784,158.140
C01205=1029.902,7.044,-91.784,168.052,43.782,158.140
C01206=1029.909,7.294,-91.799,168.055,43.780,158.140
C01207=1029.915,7.543,-91.814,168.058,43.779,158.140
C01208=1029.921,7.793,-91.829,168.060,43.777,158.140
C01209=1029.928,8.043,-91.844,168.063,43.775,158.139
C01210=1029.934,8.292,-91.859,168.065,43.774,158.139
C01211=1029.940,8.541,-91.874,168.067,43.772,158.139
C01212=1029.946,8.791,-91.889,168.070,43.770,158.139
C01213=1029.953,9.041,-91.903,168.073,43.769,158.139
C01214=1029.959,9.290,-91.919,168.075,43.767,158.139
C01215=1029.965,9.539,-91.934,168.078,43.765,158.139
C01216=1029.972,9.788,-91.949,168.080,43.764,158.139
C01217=1029.978,10.038,-91.964,168.082,43.762,158.139
C01218=1029.984,10.288,-91.979,168.085,43.761,158.139
C01219=1029.991,10.537,-91.993,168.088,43.759,158.138
C01220=1029.997,10.787,-92.008,168.090,43.757,158.138
C01221=1030.004,11.036,-92.024,168.092,43.755,158.138
C01222=1030.010,11.285,-92.039,168.095,43.754,158.138
C01223=1030.017,11.570,-92.056,168.097,43.752,158.138
C01224=1030.024,11.855,-92.073,168.101,43.750,158.138
C01225=1030.031,12.140,-92.091,168.104,43.748,158.138
C01226=1030.039,12.425,-92.107,168.106,43.746,158.138
C01227=1030.045,12.674,-92.122,168.109,43.744,158.138
C01228=1030.052,12.924,-92.137,168.112,43.742,158.137
C01229=1030.058,13.173,-92.153,168.113,43.741,158.137
C01230=1030.063,13.422,-92.168,168.116,43.739,158.137
C01231=1030.070,13.672,-92.183,168.119,43.738,158.137
C01232=1030.076,13.922,-92.198,168.121,43.736,158.137
C01233=1030.083,14.171,-92.214,168.123,43.734,158.137
C01234=1030.089,14.420,-92.229,168.126,43.733,158.137
C01235=1030.095,14.670,-92.244,168.128,43.731,158.137
C01236=1030.102,14.919,-92.260,168.131,43.730,158.137
C01237=1030.108,15.169,-92.275,168.133,43.728,158.137
C01238=1030.114,15.419,-92.290,168.135,43.726,158.136
C01239=1030.120,15.668,-92.306,168.138,43.725,158.137
C01240=1030.127,15.918,-92.321,168.141,43.723,158.136
C01241=1030.133,16.167,-92.336,168.142,43.721,158.136
C01242=1030.138,16.416,-92.352,168.145,43.720,158.136
C01243=1030.145,16.666,-92.367,168.148,43.718,158.136
C01244=1030.152,16.915,-92.382,168.150,43.716,158.136
C01245=1030.158,17.164,-92.397,168.152,43.715,158.136
C01246=1030.164,17.414,-92.414,168.155,43.713,158.136
C01247=1030.170,17.663,-92.428,168.158,43.712,158.136
C01248=1030.177,17.913,-92.443,168.160,43.710,158.136
C01249=1030.183,18.162,-92.460,168.162,43.709,158.135
C01250=1030.189,18.412,-92.475,168.165,43.707,158.135
C01251=1030.196,18.661,-92.490,168.167,43.705,158.135
C01252=1030.201,18.911,-92.506,168.170,43.704,158.135
C01253=1030.208,19.160,-92.521,168.172,43.702,158.135
C01254=1030.214,19.410,-92.536,168.175,43.701,158.135
C01255=1030.221,19.659,-92.552,168.177,43.699,158.135
C01256=1030.227,19.909,-92.568,168.179,43.698,158.135
C01257=1030.233,20.158,-92.583,168.182,43.696,158.135
C01258=1030.239,20.408,-92.599,168.184,43.694,158.135
C01259=1030.246,20.657,-92.614,168.187,43.693,158.135
C01260=1030.251,20.907,-92.630,168.189,43.691,158.134
C01261=1030.258,21.156,-92.646,168.191,43.690,158.135
C01262=1030.264,21.405,-92.662,168.194,43.688,158.134
C01263=1030.270,21.655,-92.677,168.196,43.686,158.134
C01264=1030.277,21.904,-92.693,168.199,43.685,158.134
C01265=1030.283,22.154,-92.708,168.201,43.683,158.134
C01266=1030.289,22.403,-92.724,168.204,43.681,158.134
C01267=1030.295,22.653,-92.739,168.206,43.680,158.134
C01268=1030.302,22.902,-92.755,168.208,43.678,158.134
C01269=1030.308,23.151,-92.771,168.211,43.677,158.134
C01270=1030.314,23.401,-92.786,168.213,43.676,158.134
C01271=1030.320,23.650,-92.802,168.215,43.674,158.133
C01272=1030.327,23.899,-92.818,168.218,43.672,158.133
C01273=1030.332,24.149,-92.834,168.221,43.671,158.133
C01274=1030.339,24.398,-92.849,168.222,43.669,158.133
C01275=1030.346,24.647,-92.865,168.225,43.668,158.133
C01276=1030.351,24.897,-92.880,168.228,43.666,158.133
C01277=1030.358,25.146,-92.896,168.229,43.664,158.133
C01278=1030.364,25.396,-92.912,168.232,43.663,158.133
C01279=1030.371,25.646,-92.928,168.235,43.661,158.133
C01280=1030.377,25.895,-92.944,168.238,43.659,158.133
C01281=1030.384,26.144,-92.960,168.239,43.658,158.133
C01282=1030.390,26.394,-92.976,168.242,43.656,158.132
C01283=1030.396,26.643,-92.991,168.245,43.654,158.132
C01284=1030.402,26.893,-93.007,168.246,43.653,158.132
C01285=1030.409,27.142,-93.023,168.249,43.651,158.132
C01286=1030.415,27.391,-93.039,168.252,43.650,158.132
C01287=1030.422,27.678,-93.057,168.255,43.648,158.132
C01288=1030.429,27.963,-93.075,168.257,43.646,158.132
C01289=1030.437,28.249,-93.093,168.260,43.645,158.132
C01290=1030.444,28.536,-93.112,168.262,43.643,158.132
C01291=1030.450,28.786,-93.127,168.265,43.641,158.132
C01292=1030.456,29.035,-93.144,168.267,43.640,158.131
C01293=1030.462,29.284,-93.159,168.269,43.638,158.131
C01294=1030.468,29.533,-93.176,168.272,43.637,158.131
C01295=1030.474,29.783,-93.192,168.274,43.635,158.131
C01296=1030.480,30.032,-93.208,168.277,43.634,158.131
C01297=1030.487,30.281,-93.224,168.279,43.632,158.131
C01298=1030.493,30.530,-93.240,168.281,43.630,158.131
C01299=1030.499,30.780,-93.257,168.284,43.629,158.131
C01300=1030.506,31.030,-93.272,168.286,43.627,158.131
C01301=1030.512,31.279,-93.288,168.289,43.626,158.131
C01302=1030.518,31.529,-93.304,168.291,43.624,158.131
C01303=1030.524,31.778,-93.320,168.294,43.623,158.131
C01304=1030.530,32.027,-93.336,168.296,43.621,158.130
C01305=1030.537,32.277,-93.353,168.298,43.619,158.130
C01306=1030.543,32.527,-93.369,168.301,43.618,158.130
C01307=1030.549,32.776,-93.385,168.303,43.616,158.130
C01308=1030.555,33.025,-93.401,168.305,43.615,158.130
C01309=1030.561,33.274,-93.417,168.308,43.613,158.130
C01310=1030.568,33.523,-93.433,168.310,43.612,158.130
C01311=1030.575,33.773,-93.449,168.312,43.611,158.130
C01312=1030.581,34.023,-93.466,168.315,43.609,158.130
C01313=1030.587,34.272,-93.481,168.318,43.607,158.130
C01314=1030.593,34.521,-93.498,168.319,43.606,158.129
C01315=1030.599,34.770,-93.514,168.322,43.604,158.129
C01316=1030.606,35.021,-93.530,168.325,43.602,158.129
C01317=1030.612,35.270,-93.546,168.326,43.601,158.129
C01318=1030.618,35.519,-93.562,168.329,43.599,158.129
C01319=1030.624,35.768,-93.579,168.332,43.598,158.129
C01320=1030.631,36.018,-93.595,168.333,43.596,158.129
C01321=1030.638,36.267,-93.611,168.336,43.594,158.129
C01322=1030.643,36.517,-93.627,168.339,43.593,158.129
C01323=1030.650,36.765,-93.644,168.341,43.591,158.129
C01324=1030.657,37.015,-93.660,168.343,43.590,158.128
C01325=1030.663,37.265,-93.676,168.346,43.588,158.128
C01326=1030.669,37.514,-93.693,168.348,43.587,158.128
C01327=1030.675,37.763,-93.709,168.350,43.585,158.128
C01328=1030.681,38.013,-93.726,168.353,43.584,158.128
C01329=1030.687,38.263,-93.742,168.355,43.583,158.128
C01330=1030.694,38.511,-93.759,168.358,43.581,158.128
C01331=1030.700,38.761,-93.775,168.360,43.579,158.128
C01332=1030.706,39.010,-93.791,168.362,43.578,158.128
C01333=1030.712,39.260,-93.808,168.365,43.576,158.128
C01334=1030.718,39.509,-93.824,168.366,43.575,158.128
C01335=1030.724,39.758,-93.841,168.369,43.573,158.127
C01336=1030.731,40.008,-93.858,168.372,43.572,158.127
C01337=1030.737,40.258,-93.874,168.373,43.570,158.127
C01338=1030.743,40.507,-93.890,168.376,43.569,158.127
C01339=1030.749,40.756,-93.907,168.379,43.567,158.127
C01340=1030.756,41.006,-93.924,168.381,43.565,158.127
C01341=1030.761,41.255,-93.940,168.383,43.564,158.127
C01342=1030.768,41.504,-93.957,168.386,43.562,158.127
C01343=1030.774,41.754,-93.974,168.388,43.561,158.127
C01344=1030.781,42.003,-93.989,168.390,43.559,158.127
C01345=1030.787,42.252,-94.006,168.392,43.558,158.127
C01346=1030.793,42.501,-94.023,168.395,43.557,158.127
C01347=1030.800,42.751,-94.039,168.398,43.555,158.126
C01348=1030.806,43.000,-94.055,168.399,43.554,158.126
C01349=1030.811,43.249,-94.073,168.402,43.552,158.126
C01350=1030.818,43.499,-94.090,168.405,43.551,158.126
C01351=1030.825,43.785,-94.110,168.407,43.549,158.126
C01352=1030.832,44.071,-94.128,168.409,43.548,158.126
C01353=1030.838,44.357,-94.147,168.412,43.546,158.126
C01354=1030.846,44.643,-94.167,168.415,43.544,158.126
C01355=1030.851,44.893,-94.183,168.417,43.543,158.126
C01356=1030.858,45.142,-94.201,168.420,43.542,158.126
C01357=1030.864,45.392,-94.217,168.422,43.540,158.126
C01358=1030.870,45.640,-94.234,168.425,43.539,158.126
C01359=1030.876,45.891,-94.251,168.426,43.537,158.125
C01360=1030.882,46.139,-94.268,168.429,43.536,158.125
C01361=1030.888,46.389,-94.284,168.432,43.534,158.125
C01362=1030.895,46.638,-94.302,168.434,43.533,158.125
C01363=1030.901,46.887,-94.318,168.436,43.531,158.125
C01364=1030.907,47.136,-94.336,168.438,43.530,158.125
C01365=1030.913,47.387,-94.352,168.441,43.528,158.125
C01366=1030.919,47.635,-94.369,168.443,43.527,158.125
C01367=1030.925,47.885,-94.385,168.445,43.525,158.125
C01368=1030.931,48.134,-94.403,168.448,43.524,158.125
C01369=1030.937,48.384,-94.420,168.450,43.522,158.125
C01370=1030.944,48.633,-94.437,168.452,43.521,158.125
C01371=1030.950,48.882,-94.454,168.454,43.519,158.124
C01372=1030.956,49.132,-94.471,168.457,43.518,158.124
C01373=1030.963,49.381,-94.488,168.459,43.516,158.124
C01374=1030.968,49.630,-94.504,168.461,43.515,158.124
C01375=1030.975,49.880,-94.522,168.464,43.514,158.124
C01376=1030.981,50.129,-94.539,168.467,43.512,158.124
C01377=1030.987,50.378,-94.555,168.468,43.511,158.124
C01378=1030.994,50.628,-94.573,168.471,43.509,158.124
C01379=1030.999,50.877,-94.590,168.473,43.508,158.124
C01380=1031.006,51.127,-94.607,168.476,43.507,158.124
C01381=1031.012,51.375,-94.624,168.478,43.505,158.124
C01382=1031.018,51.625,-94.640,168.480,43.504,158.124
C01383=1031.024,51.874,-94.658,168.483,43.502,158.123
C01384=1031.030,52.123,-94.675,168.484,43.501,158.123
C01385=1031.037,52.373,-94.692,168.487,43.499,158.123
C01386=1031.043,52.622,-94.709,168.490,43.498,158.123
C01387=1031.049,52.872,-94.727,168.492,43.496,158.123
C01388=1031.055,53.121,-94.743,168.494,43.494,158.123
C01389=1031.062,53.370,-94.760,168.496,43.493,158.123
C01390=1031.068,53.619,-94.777,168.499,43.491,158.123
C01391=1031.074,53.870,-94.794,168.501,43.490,158.123
C01392=1031.080,54.118,-94.811,168.503,43.488,158.123
C01393=1031.087,54.368,-94.829,168.506,43.487,158.123
C01394=1031.092,54.617,-94.846,168.508,43.486,158.122
C01395=1031.099,54.867,-94.863,168.510,43.484,158.122
C01396=1031.106,55.116,-94.880,168.513,43.483,158.122
C01397=1031.112,55.365,-94.897,168.515,43.481,158.122
C01398=1031.118,55.615,-94.914,168.517,43.480,158.122
C01399=1031.125,55.864,-94.931,168.520,43.478,158.122
C01400=1031.131,56.113,-94.948,168.522,43.477,158.122
C01401=1031.137,56.363,-94.966,168.525,43.475,158.122
C01402=1031.143,56.612,-94.983,168.526,43.473,158.122
C01403=1031.150,56.861,-95.000,168.529,43.472,158.122
C01404=1031.156,57.110,-95.017,168.532,43.470,158.121
C01405=1031.162,57.360,-95.035,168.533,43.469,158.121
C01406=1031.168,57.609,-95.052,168.536,43.467,158.121
C01407=1031.175,57.859,-95.068,168.539,43.465,158.121
C01408=1031.180,58.108,-95.086,168.540,43.464,158.121
C01409=1031.187,58.357,-95.103,168.543,43.463,158.121
C01410=1031.194,58.606,-95.121,168.545,43.462,158.121
C01411=1031.200,58.856,-95.138,168.548,43.460,158.121
C01412=1031.207,59.105,-95.156,168.550,43.458,158.121
C01413=1031.212,59.354,-95.172,168.552,43.457,158.121
C01414=1031.219,59.604,-95.189,168.555,43.455,158.120
C01415=1031.226,59.890,-95.209,168.557,43.453,158.120
C01416=1031.234,60.175,-95.230,168.560,43.451,158.120
C01417=1031.241,60.461,-95.249,168.563,43.449,158.120
C01418=1031.248,60.747,-95.269,168.565,43.448,158.120
C01419=1031.254,60.995,-95.286,168.568,43.446,158.120
C01420=1031.261,61.245,-95.304,168.570,43.445,158.120
C01421=1031.267,61.495,-95.321,168.572,43.443,158.120
C01422=1031.273,61.744,-95.338,168.575,43.442,158.120
C01423=1031.280,61.993,-95.355,168.577,43.440,158.119
C01424=1031.286,62.243,-95.373,168.579,43.439,158.119
C01425=1031.293,62.492,-95.390,168.582,43.437,158.119
C01426=1031.299,62.741,-95.407,168.584,43.435,158.119
C01427=1031.305,62.990,-95.425,168.587,43.434,158.119
C01428=1031.312,63.240,-95.442,168.589,43.432,158.119
C01429=1031.319,63.489,-95.459,168.591,43.430,158.119
C01430=1031.324,63.738,-95.477,168.594,43.429,158.119
C01431=1031.330,63.988,-95.495,168.595,43.428,158.118
C01432=1031.337,64.237,-95.512,168.598,43.426,158.118
C01433=1031.343,64.486,-95.530,168.601,43.425,158.118
C01434=1031.350,64.736,-95.547,168.603,43.424,158.118
C01435=1031.356,64.985,-95.565,168.605,43.422,158.118
C01436=1031.361,65.234,-95.583,168.607,43.421,158.118
C01437=1031.368,65.483,-95.601,168.610,43.419,158.118
C01438=1031.374,65.732,-95.618,168.612,43.418,158.118
C01439=1031.381,65.982,-95.636,168.614,43.416,158.118
C01440=1031.387,66.231,-95.654,168.617,43.415,158.118
C01441=1031.392,66.481,-95.671,168.619,43.413,158.118
C01442=1031.399,66.730,-95.688,168.621,43.412,158.118
C01443=1031.405,66.980,-95.706,168.623,43.410,158.117
C01444=1031.412,67.228,-95.724,168.626,43.409,158.117
C01445=1031.418,67.478,-95.742,168.628,43.407,158.117
C01446=1031.424,67.727,-95.760,168.630,43.406,158.117
C01447=1031.430,67.976,-95.777,168.633,43.404,158.117
C01448=1031.437,68.226,-95.795,168.634,43.403,158.117
C01449=1031.443,68.475,-95.814,168.637,43.401,158.117
C01450=1031.449,68.724,-95.831,168.640,43.400,158.117
C01451=1031.455,68.973,-95.848,168.642,43.399,158.117
C01452=1031.462,69.223,-95.866,168.644,43.397,158.117
C01453=1031.468,69.473,-95.884,168.646,43.396,158.117
C01454=1031.474,69.721,-95.902,168.649,43.394,158.117
C01455=1031.480,69.971,-95.920,168.652,43.393,158.116
C01456=1031.486,70.220,-95.938,168.654,43.392,158.116
C01457=1031.492,70.469,-95.956,168.656,43.390,158.116
C01458=1031.498,70.719,-95.974,168.658,43.389,158.116
C01459=1031.505,70.968,-95.991,168.661,43.387,158.116
C01460=1031.511,71.217,-96.009,168.662,43.386,158.116
C01461=1031.517,71.466,-96.028,168.665,43.384,158.116
C01462=1031.523,71.716,-96.046,168.668,43.383,158.116
C01463=1031.529,71.966,-96.063,168.669,43.381,158.116
C01464=1031.535,72.214,-96.082,168.672,43.380,158.116
C01465=1031.542,72.464,-96.099,168.674,43.378,158.115
C01466=1031.549,72.713,-96.118,168.677,43.377,158.115
C01467=1031.554,72.962,-96.135,168.678,43.375,158.115
C01468=1031.560,73.211,-96.153,168.681,43.374,158.115
C01469=1031.567,73.461,-96.172,168.684,43.372,158.115
C01470=1031.573,73.710,-96.190,168.686,43.371,158.115
C01471=1031.579,73.959,-96.207,168.688,43.370,158.115
C01472=1031.585,74.208,-96.225,168.690,43.369,158.115
C01473=1031.592,74.458,-96.243,168.693,43.367,158.115
C01474=1031.598,74.707,-96.262,168.696,43.366,158.115
C01475=1031.604,74.957,-96.280,168.697,43.364,158.115
C01476=1031.610,75.205,-96.298,168.700,43.363,158.115
C01477=1031.617,75.455,-96.316,168.702,43.361,158.114
C01478=1031.623,75.704,-96.334,168.704,43.360,158.114
C01479=1031.630,75.990,-96.354,168.707,43.358,158.114
C01480=1031.637,76.275,-96.375,168.710,43.356,158.114
C01481=1031.644,76.561,-96.396,168.713,43.355,158.114
C01482=1031.651,76.846,-96.417,168.715,43.353,158.114
C01483=1031.657,77.096,-96.435,168.717,43.351,158.114
C01484=1031.664,77.345,-96.453,168.720,43.350,158.114
C01485=1031.670,77.594,-96.471,168.722,43.349,158.114
C01486=1031.676,77.844,-96.490,168.724,43.347,158.114
C01487=1031.682,78.092,-96.508,168.727,43.346,158.114
C01488=1031.688,78.342,-96.526,168.729,43.344,158.113
C01489=1031.695,78.591,-96.545,168.731,43.343,158.113
C01490=1031.701,78.841,-96.563,168.733,43.342,158.113
C01491=1031.707,79.090,-96.581,168.736,43.340,158.113
C01492=1031.712,79.338,-96.600,168.738,43.339,158.113
C01493=1031.718,79.588,-96.618,168.740,43.338,158.113
C01494=1031.725,79.837,-96.637,168.743,43.336,158.113
C01495=1031.731,80.086,-96.656,168.745,43.335,158.113
C01496=1031.737,80.336,-96.673,168.748,43.334,158.113
C01497=1031.744,80.585,-96.692,168.749,43.333,158.113
C01498=1031.750,80.834,-96.710,168.752,43.331,158.113
C01499=1031.756,81.083,-96.728,168.754,43.330,158.113
C01500=1031.761,81.333,-96.748,168.756,43.328,158.112
C01501=1031.768,81.582,-96.766,168.759,43.327,158.112
C01502=1031.774,81.832,-96.784,168.761,43.326,158.112
C01503=1031.780,82.081,-96.803,168.764,43.324,158.112
C01504=1031.786,82.329,-96.821,168.766,43.323,158.112
C01505=1031.792,82.579,-96.839,168.768,43.321,158.112
C01506=1031.799,82.828,-96.858,168.770,43.320,158.112
C01507=1031.805,83.077,-96.876,168.773,43.318,158.112
C01508=1031.811,83.327,-96.896,168.776,43.317,158.112
C01509=1031.817,83.576,-96.913,168.777,43.316,158.112
C01510=1031.823,83.826,-96.932,168.780,43.314,158.112
C01511=1031.830,84.075,-96.951,168.782,43.313,158.112
C01512=1031.836,84.323,-96.969,168.784,43.311,158.111
C01513=1031.842,84.573,-96.987,168.787,43.310,158.111
C01514=1031.848,84.822,-97.006,168.789,43.308,158.111
C01515=1031.855,85.071,-97.024,168.792,43.307,158.111
C01516=1031.860,85.321,-97.044,168.793,43.306,158.111
C01517=1031.867,85.570,-97.062,168.796,43.304,158.111
C01518=1031.873,85.819,-97.080,168.798,43.303,158.111
C01519=1031.879,86.069,-97.099,168.801,43.301,158.111
C01520=1031.886,86.318,-97.117,168.803,43.300,158.111
C01521=1031.892,86.567,-97.136,168.805,43.299,158.111
C01522=1031.899,86.816,-97.155,168.808,43.297,158.111
C01523=1031.904,87.066,-97.173,168.810,43.296,158.110
C01524=1031.910,87.315,-97.192,168.812,43.295,158.110
C01525=1031.916,87.563,-97.210,168.815,43.293,158.110
C01526=1031.923,87.813,-97.229,168.817,43.292,158.110
C01527=1031.929,88.062,-97.247,168.819,43.290,158.110
C01528=1031.936,88.311,-97.266,168.821,43.289,158.110
C01529=1031.941,88.560,-97.285,168.824,43.287,158.110
C01530=1031.948,88.809,-97.304,168.827,43.286,158.110
C01531=1031.954,89.059,-97.322,168.828,43.284,158.110
C01532=1031.960,89.308,-97.341,168.831,43.283,158.110
C01533=1031.967,89.557,-97.359,168.834,43.281,158.110
C01534=1031.973,89.807,-97.378,168.836,43.280,158.110
C01535=1031.979,90.056,-97.397,168.838,43.278,158.109
C01536=1031.985,90.305,-97.416,168.840,43.277,158.109
C01537=1031.991,90.555,-97.435,168.843,43.276,158.109
C01538=1031.997,90.804,-97.454,168.845,43.275,158.109
C01539=1032.003,91.053,-97.473,168.847,43.273,158.109
C01540=1032.009,91.302,-97.492,168.850,43.272,158.109
C01541=1032.016,91.551,-97.510,168.852,43.270,158.109
C01542=1032.022,91.801,-97.529,168.855,43.269,158.109
C01543=1032.028,92.086,-97.551,168.857,43.267,158.109
C01544=1032.036,92.371,-97.574,168.860,43.266,158.109
C01545=1032.042,92.657,-97.595,168.862,43.265,158.109
C01546=1032.050,92.942,-97.616,168.865,43.263,158.109
C01547=1032.056,93.191,-97.636,168.867,43.262,158.108
C01548=1032.062,93.440,-97.654,168.870,43.260,158.108
C01549=1032.068,93.690,-97.674,168.872,43.259,158.108
C01550=1032.074,93.939,-97.692,168.874,43.258,158.108
C01551=1032.080,94.188,-97.711,168.876,43.257,158.108
C01552=1032.087,94.438,-97.730,168.879,43.255,158.108
C01553=1032.093,94.688,-97.750,168.882,43.254,158.108
C01554=1032.099,94.936,-97.769,168.884,43.253,158.108
C01555=1032.106,95.185,-97.788,168.886,43.251,158.108
C01556=1032.111,95.435,-97.807,168.888,43.250,158.108
C01557=1032.118,95.684,-97.826,168.891,43.248,158.108
C01558=1032.123,95.933,-97.845,168.894,43.247,158.108
C01559=1032.130,96.182,-97.863,168.895,43.246,158.108
C01560=1032.136,96.431,-97.883,168.898,43.244,158.107
C01561=1032.142,96.680,-97.902,168.900,43.243,158.107
C01562=1032.148,96.930,-97.921,168.902,43.241,158.107
C01563=1032.154,97.179,-97.940,168.905,43.240,158.107
C01564=1032.160,97.428,-97.959,168.907,43.239,158.107
C01565=1032.167,97.677,-97.979,168.910,43.237,158.107
C01566=1032.173,97.926,-97.998,168.912,43.236,158.107
C01567=1032.179,98.175,-98.016,168.914,43.234,158.107
C01568=1032.185,98.425,-98.036,168.917,43.233,158.107
C01569=1032.192,98.674,-98.055,168.919,43.232,158.107
C01570=1032.198,98.923,-98.074,168.921,43.230,158.107
C01571=1032.204,99.172,-98.093,168.923,43.229,158.107
C01572=1032.211,99.422,-98.112,168.926,43.227,158.106
C01573=1032.217,99.670,-98.132,168.929,43.226,158.106
C01574=1032.223,99.919,-98.151,168.930,43.224,158.106
C01575=1032.229,100.169,-98.170,168.933,43.223,158.106
C01576=1032.235,100.418,-98.190,168.935,43.222,158.106
C01577=1032.241,100.668,-98.209,168.938,43.220,158.106
C01578=1032.247,100.917,-98.228,168.940,43.219,158.106
C01579=1032.253,101.166,-98.248,168.942,43.218,158.106
C01580=1032.259,101.415,-98.267,168.945,43.217,158.106
C01581=1032.266,101.664,-98.287,168.947,43.215,158.106
C01582=1032.271,101.913,-98.306,168.950,43.214,158.106
C01583=1032.277,102.163,-98.325,168.951,43.213,158.106
C01584=1032.283,102.411,-98.345,168.954,43.211,158.106
C01585=1032.290,102.661,-98.364,168.957,43.210,158.106
C01586=1032.296,102.910,-98.384,168.959,43.209,158.106
C01587=1032.302,103.160,-98.403,168.961,43.207,158.105
C01588=1032.308,103.408,-98.423,168.963,43.206,158.105
C01589=1032.314,103.657,-98.442,168.966,43.205,158.105
C01590=1032.320,103.906,-98.462,168.969,43.204,158.105
C01591=1032.326,104.156,-98.481,168.970,43.202,158.105
C01592=1032.333,104.405,-98.501,168.973,43.201,158.105
C01593=1032.339,104.654,-98.520,168.975,43.200,158.105
C01594=1032.345,104.903,-98.540,168.978,43.198,158.105
C01595=1032.351,105.153,-98.559,168.981,43.197,158.105
C01596=1032.357,105.401,-98.579,168.982,43.196,158.105
C01597=1032.362,105.651,-98.598,168.985,43.194,158.105
C01598=1032.370,105.900,-98.618,168.987,43.193,158.105
C01599=1032.375,106.149,-98.637,168.990,43.192,158.105
C01600=1032.381,106.398,-98.657,168.992,43.190,158.104
C01601=1032.387,106.648,-98.677,168.994,43.189,158.104
C01602=1032.394,106.896,-98.696,168.997,43.188,158.104
C01603=1032.400,107.146,-98.716,169.000,43.186,158.104
C01604=1032.406,107.395,-98.736,169.001,43.185,158.104
C01605=1032.412,107.644,-98.756,169.004,43.184,158.104
C01606=1032.418,107.893,-98.774,169.006,43.183,158.104
C01607=1032.425,108.179,-98.797,169.009,43.181,158.104
C01608=1032.433,108.464,-98.820,169.011,43.180,158.104
C01609=1032.440,108.749,-98.842,169.015,43.178,158.104
C01610=1032.447,109.035,-98.865,169.018,43.176,158.104
C01611=1032.453,109.284,-98.884,169.020,43.175,158.104
C01612=1032.459,109.533,-98.904,169.022,43.174,158.104
C01613=1032.465,109.783,-98.924,169.024,43.173,158.103
C01614=1032.471,110.031,-98.944,169.027,43.171,158.103
C01615=1032.478,110.281,-98.963,169.030,43.170,158.103
C01616=1032.484,110.530,-98.983,169.031,43.169,158.103
C01617=1032.490,110.779,-99.003,169.034,43.167,158.103
C01618=1032.496,111.028,-99.022,169.037,43.166,158.103
C01619=1032.502,111.277,-99.042,169.039,43.165,158.103
C01620=1032.509,111.527,-99.062,169.042,43.163,158.103
C01621=1032.515,111.775,-99.082,169.043,43.162,158.103
C01622=1032.520,112.025,-99.102,169.046,43.161,158.103
C01623=1032.526,112.274,-99.122,169.049,43.159,158.103
C01624=1032.533,112.523,-99.142,169.051,43.158,158.103
C01625=1032.539,112.772,-99.162,169.053,43.157,158.103
C01626=1032.545,113.021,-99.181,169.056,43.155,158.103
C01627=1032.551,113.271,-99.201,169.058,43.154,158.103
C01628=1032.557,113.520,-99.221,169.061,43.153,158.103
C01629=1032.563,113.769,-99.241,169.063,43.152,158.103
C01630=1032.569,114.018,-99.262,169.065,43.150,158.102
C01631=1032.575,114.267,-99.282,169.068,43.149,158.102
C01632=1032.581,114.516,-99.302,169.070,43.148,158.102
C01633=1032.587,114.765,-99.322,169.073,43.147,158.102
C01634=1032.593,115.014,-99.342,169.075,43.146,158.102
C01635=1032.599,115.264,-99.362,169.077,43.145,158.102
C01636=1032.605,115.513,-99.382,169.080,43.143,158.102
C01637=1032.611,115.762,-99.402,169.082,43.142,158.102
C01638=1032.617,116.011,-99.423,169.085,43.141,158.102
C01639=1032.623,116.260,-99.443,169.087,43.140,158.102
C01640=1032.629,116.509,-99.463,169.089,43.139,158.102
C01641=1032.635,116.759,-99.483,169.092,43.138,158.102
C01642=1032.641,117.008,-99.503,169.094,43.136,158.102
C01643=1032.647,117.256,-99.523,169.097,43.135,158.102
C01644=1032.652,117.505,-99.544,169.098,43.134,158.102
C01645=1032.659,117.755,-99.564,169.101,43.133,158.102
C01646=1032.665,118.004,-99.584,169.104,43.131,158.102
C01647=1032.671,118.253,-99.604,169.106,43.130,158.102
C01648=1032.677,118.502,-99.625,169.109,43.129,158.101
C01649=1032.683,118.751,-99.645,169.111,43.128,158.101
C01650=1032.689,119.001,-99.665,169.113,43.127,158.101
C01651=1032.695,119.250,-99.685,169.116,43.125,158.101
C01652=1032.701,119.498,-99.707,169.119,43.124,158.101
C01653=1032.708,119.748,-99.727,169.121,43.123,158.101
C01654=1032.714,119.996,-99.747,169.123,43.121,158.101
C01655=1032.720,120.245,-99.767,169.125,43.120,158.101
C01656=1032.725,120.495,-99.788,169.128,43.119,158.101
C01657=1032.731,120.744,-99.808,169.131,43.118,158.101
C01658=1032.737,120.993,-99.828,169.133,43.117,158.101
C01659=1032.744,121.242,-99.848,169.135,43.115,158.101
C01660=1032.749,121.491,-99.869,169.138,43.114,158.101
C01661=1032.756,121.741,-99.889,169.140,43.113,158.101
C01662=1032.762,121.989,-99.910,169.143,43.112,158.101
C01663=1032.769,122.239,-99.930,169.146,43.111,158.101
C01664=1032.774,122.488,-99.950,169.147,43.109,158.101
C01665=1032.780,122.736,-99.970,169.150,43.108,158.101
C01666=1032.787,122.986,-99.991,169.153,43.107,158.101
C01667=1032.793,123.235,-100.011,169.155,43.106,158.101
C01668=1032.799,123.484,-100.032,169.157,43.104,158.100
C01669=1032.805,123.733,-100.052,169.160,43.103,158.100
C01670=1032.811,123.982,-100.073,169.162,43.102,158.100
C01671=1032.818,124.267,-100.096,169.165,43.101,158.100
C01672=1032.825,124.552,-100.120,169.169,43.099,158.100
C01673=1032.832,124.837,-100.143,169.171,43.097,158.100
C01674=1032.839,125.123,-100.166,169.174,43.096,158.100
C01675=1032.845,125.372,-100.187,169.176,43.095,158.100
C01676=1032.851,125.622,-100.207,169.179,43.093,158.100
C01677=1032.857,125.870,-100.227,169.182,43.092,158.100
C01678=1032.864,126.120,-100.247,169.183,43.091,158.100
C01679=1032.869,126.368,-100.269,169.186,43.089,158.100
C01680=1032.876,126.618,-100.289,169.189,43.088,158.100
C01681=1032.882,126.867,-100.309,169.192,43.087,158.100
C01682=1032.889,127.116,-100.330,169.194,43.086,158.100
C01683=1032.894,127.365,-100.351,169.196,43.084,158.100
C01684=1032.901,127.614,-100.371,169.199,43.083,158.100
C01685=1032.907,127.864,-100.391,169.201,43.082,158.099
C01686=1032.913,128.112,-100.412,169.204,43.081,158.099
C01687=1032.920,128.362,-100.433,169.206,43.079,158.099
C01688=1032.926,128.611,-100.453,169.209,43.078,158.099
C01689=1032.932,128.859,-100.474,169.211,43.077,158.099
C01690=1032.938,129.109,-100.494,169.214,43.076,158.099
C01691=1032.945,129.357,-100.515,169.216,43.074,158.099
C01692=1032.951,129.606,-100.535,169.218,43.073,158.099
C01693=1032.956,129.856,-100.556,169.221,43.072,158.099
C01694=1032.963,130.104,-100.577,169.224,43.071,158.099
C01695=1032.969,130.354,-100.597,169.227,43.069,158.099
C01696=1032.976,130.603,-100.618,169.228,43.068,158.099
C01697=1032.982,130.852,-100.639,169.231,43.067,158.099
C01698=1032.987,131.102,-100.660,169.234,43.066,158.099
C01699=1032.994,131.350,-100.680,169.236,43.065,158.099
C01700=1033.000,131.600,-100.701,169.239,43.063,158.099
C01701=1033.006,131.848,-100.722,169.242,43.062,158.099
C01702=1033.012,132.098,-100.743,169.244,43.061,158.099
C01703=1033.018,132.347,-100.765,169.246,43.060,158.099
C01704=1033.024,132.595,-100.785,169.249,43.059,158.099
C01705=1033.030,132.845,-100.806,169.252,43.057,158.098
C01706=1033.036,133.093,-100.827,169.253,43.056,158.098
C01707=1033.042,133.343,-100.848,169.256,43.055,158.098
C01708=1033.048,133.591,-100.869,169.259,43.054,158.098
C01709=1033.054,133.841,-100.889,169.261,43.053,158.098
C01710=1033.060,134.090,-100.911,169.264,43.052,158.098
C01711=1033.067,134.338,-100.932,169.267,43.051,158.098
C01712=1033.073,134.588,-100.953,169.270,43.049,158.098
C01713=1033.078,134.837,-100.974,169.271,43.048,158.098
C01714=1033.085,135.086,-100.995,169.274,43.047,158.098
C01715=1033.091,135.335,-101.016,169.277,43.046,158.098
C01716=1033.097,135.584,-101.037,169.280,43.044,158.098
C01717=1033.103,135.833,-101.057,169.281,43.043,158.098
C01718=1033.109,136.082,-101.079,169.284,43.042,158.098
C01719=1033.116,136.331,-101.100,169.287,43.041,158.098
C01720=1033.121,136.581,-101.121,169.289,43.040,158.098
C01721=1033.127,136.829,-101.142,169.292,43.039,158.098
C01722=1033.134,137.078,-101.163,169.295,43.038,158.098
C01723=1033.140,137.327,-101.185,169.297,43.036,158.098
C01724=1033.145,137.576,-101.205,169.299,43.035,158.098
C01725=1033.151,137.826,-101.227,169.302,43.034,158.098
C01726=1033.158,138.074,-101.248,169.305,43.033,158.098
C01727=1033.164,138.323,-101.269,169.308,43.032,158.098
C01728=1033.170,138.573,-101.290,169.310,43.031,158.098
C01729=1033.177,138.822,-101.311,169.312,43.030,158.098
C01730=1033.182,139.070,-101.332,169.315,43.029,158.098
C01731=1033.188,139.319,-101.354,169.318,43.028,158.098
C01732=1033.194,139.568,-101.375,169.320,43.027,158.098
C01733=1033.200,139.818,-101.396,169.323,43.025,158.098
C01734=1033.206,140.067,-101.418,169.326,43.024,158.098
C01735=1033.213,140.352,-101.442,169.328,43.022,158.097
C01736=1033.220,140.637,-101.467,169.331,43.021,158.097
C01737=1033.227,140.922,-101.491,169.334,43.020,158.097
C01738=1033.233,141.207,-101.516,169.337,43.019,158.097
C01739=1033.240,141.456,-101.537,169.340,43.018,158.097
C01740=1033.246,141.705,-101.558,169.342,43.017,158.097
C01741=1033.252,141.954,-101.580,169.345,43.015,158.097
C01742=1033.258,142.203,-101.601,169.347,43.015,158.097
C01743=1033.264,142.428,-101.620,169.350,43.013,158.097
C01744=1033.269,142.653,-101.640,169.352,43.012,158.097
C01745=1033.275,142.878,-101.659,169.355,43.012,158.097
C01746=1033.280,143.102,-101.679,169.357,43.011,158.097
C01747=1033.286,143.327,-101.698,169.359,43.010,158.097
C01748=1033.291,143.552,-101.718,169.361,43.009,158.097
C01749=1033.296,143.776,-101.736,169.364,43.008,158.097
C01750=1033.302,144.001,-101.757,169.366,43.007,158.097
C01751=1033.309,144.250,-101.778,169.369,43.005,158.097
C01752=1033.314,144.499,-101.799,169.372,43.004,158.097
C01753=1033.320,144.748,-101.821,169.374,43.003,158.097
C01754=1033.327,144.997,-101.842,169.376,43.002,158.097
C01755=1033.333,145.246,-101.864,169.379,43.001,158.097
C01756=1033.338,145.495,-101.885,169.382,43.000,158.097
C01757=1033.344,145.744,-101.907,169.385,42.999,158.097
C01758=1033.351,145.993,-101.928,169.388,42.997,158.097
C01759=1033.357,146.243,-101.950,169.389,42.996,158.097
C01760=1033.364,146.491,-101.971,169.392,42.995,158.097
C01761=1033.369,146.740,-101.992,169.395,42.994,158.097
C01762=1033.375,146.990,-102.015,169.398,42.993,158.097
C01763=1033.381,147.239,-102.036,169.400,42.992,158.097
C01764=1033.387,147.488,-102.058,169.403,42.991,158.097
C01765=1033.393,147.737,-102.079,169.406,42.990,158.097
C01766=1033.399,147.985,-102.101,169.409,42.989,158.097
C01767=1033.405,148.234,-102.123,169.411,42.988,158.097
C01768=1033.411,148.483,-102.145,169.413,42.987,158.097
C01769=1033.418,148.733,-102.166,169.416,42.986,158.097
C01770=1033.424,148.982,-102.188,169.419,42.985,158.097
C01771=1033.430,149.230,-102.210,169.422,42.984,158.097
C01772=1033.436,149.479,-102.232,169.425,42.982,158.097
C01773=1033.442,149.728,-102.253,169.426,42.981,158.097
C01774=1033.447,149.978,-102.275,169.429,42.981,158.097
C01775=1033.454,150.226,-102.298,169.432,42.980,158.097
C01776=1033.459,150.475,-102.319,169.435,42.979,158.097
C01777=1033.465,150.724,-102.341,169.438,42.978,158.097
C01778=1033.472,150.973,-102.362,169.440,42.977,158.097
C01779=1033.478,151.222,-102.385,169.443,42.975,158.097
C01780=1033.484,151.471,-102.407,169.445,42.974,158.097
C01781=1033.490,151.720,-102.429,169.448,42.974,158.097
C01782=1033.496,151.969,-102.451,169.451,42.973,158.097
C01783=1033.502,152.218,-102.472,169.453,42.972,158.097
C01784=1033.508,152.467,-102.494,169.456,42.970,158.097
C01785=1033.514,152.715,-102.516,169.459,42.969,158.097
C01786=1033.520,152.965,-102.538,169.462,42.968,158.097
C01787=1033.526,153.214,-102.560,169.464,42.967,158.097
C01788=1033.532,153.463,-102.582,169.468,42.966,158.097
C01789=1033.539,153.712,-102.604,169.469,42.965,158.097
C01790=1033.545,153.961,-102.626,169.472,42.964,158.097
C01791=1033.550,154.210,-102.649,169.475,42.963,158.097
C01792=1033.557,154.459,-102.670,169.478,42.962,158.097
C01793=1033.563,154.707,-102.692,169.481,42.961,158.097
C01794=1033.569,154.956,-102.714,169.484,42.960,158.097
C01795=1033.574,155.205,-102.737,169.486,42.959,158.097
C01796=1033.581,155.454,-102.758,169.488,42.958,158.097
C01797=1033.587,155.703,-102.781,169.491,42.957,158.097
C01798=1033.592,155.952,-102.803,169.494,42.956,158.097
C01799=1033.601,156.286,-102.833,169.498,42.955,158.097
C01800=1033.609,156.619,-102.862,169.502,42.953,158.097
C01801=1033.617,156.952,-102.892,169.505,42.952,158.097
C01802=1033.626,157.285,-102.922,169.508,42.951,158.097
C01803=1033.631,157.535,-102.944,169.511,42.950,158.097
C01804=1033.638,157.783,-102.966,169.514,42.949,158.097
C01805=1033.644,158.032,-102.988,169.517,42.948,158.097
C01806=1033.649,158.281,-103.011,169.520,42.947,158.097
C01807=1033.656,158.531,-103.033,169.523,42.946,158.097
C01808=1033.662,158.779,-103.055,169.525,42.945,158.097
C01809=1033.668,159.028,-103.078,169.528,42.944,158.097
C01810=1033.674,159.277,-103.100,169.531,42.943,158.097
